LIN {X 0,Y 390.194,Z 575.883,A -85,B 0,C 180,E1 -11776.561,E2 -11776.561} C_VEL
LIN {X 0,Y 390.177,Z 575.881,A -85,B 0,C 180,E1 -11779.622,E2 -11779.622} C_VEL
LIN {X 0,Y 390.318,Z 575.868,A -85,B 0,C 180,E1 -11782.758,E2 -11782.758} C_VEL
LIN {X 0,Y 390.227,Z 575.879,A -85,B 0,C 180,E1 -11784.833,E2 -11784.833} C_VEL
LIN {X 0,Y 390.302,Z 575.869,A -85,B 0,C 180,E1 -11786.838,E2 -11786.838} C_VEL
LIN {X 0,Y 393.865,Z 588.299,A -85,B 0,C 180,E1 -11787.764,E2 -11787.764} C_VEL
LIN {X 0,Y 394.826,Z 592.713,A -85,B 0,C 180,E1 -11788.139,E2 -11788.139} C_VEL
LIN {X 0,Y 394.248,Z 604.071,A -85,B 0,C 180,E1 -11789.125,E2 -11789.125} C_VEL
LIN {X 0,Y 393.57,Z 614.626,A -85,B 0,C 180,E1 -11790.281,E2 -11790.281} C_VEL
LIN {X 0,Y 392.902,Z 623.913,A -85,B 0,C 180,E1 -11791.537,E2 -11791.537} C_VEL
LIN {X 0,Y 392.271,Z 631.723,A -85,B 0,C 180,E1 -11792.823,E2 -11792.823} C_VEL
LIN {X 0,Y 391.686,Z 639.356,A -85,B 0,C 180,E1 -11794.372,E2 -11794.372} C_VEL
LIN {X 0,Y 391.11,Z 646.386,A -85,B 0,C 180,E1 -11796.188,E2 -11796.188} C_VEL
LIN {X 0,Y 390.744,Z 651.077,A -85,B 0,C 180,E1 -11797.752,E2 -11797.752} C_VEL
LIN {X 0,Y 390.372,Z 654.695,A -85,B 0,C 180,E1 -11799.324,E2 -11799.324} C_VEL
LIN {X 0,Y 390.242,Z 656.548,A -85,B 0,C 180,E1 -11800.374,E2 -11800.374} C_VEL
LIN {X 0,Y 390.13,Z 658.928,A -85,B 0,C 180,E1 -11802.483,E2 -11802.483} C_VEL
LIN {X 0,Y 390.103,Z 659.542,A -85,B 0,C 180,E1 -11803.544,E2 -11803.544} C_VEL
LIN {X 0,Y 390.097,Z 659.724,A -85,B 0,C 180,E1 -11804.608,E2 -11804.608} C_VEL
LIN {X 0,Y 390.166,Z 659.488,A -85,B 0,C 180,E1 -11805.675,E2 -11805.675} C_VEL
LIN {X 0,Y 390.415,Z 658.214,A -85,B 0,C 180,E1 -11807.434,E2 -11807.434} C_VEL
LIN {X 0,Y 390.691,Z 656.292,A -85,B 0,C 180,E1 -11808.891,E2 -11808.891} C_VEL
LIN {X 0,Y 391.12,Z 653.303,A -85,B 0,C 180,E1 -11810.453,E2 -11810.453} C_VEL
LIN {X 0,Y 391.676,Z 648.912,A -85,B 0,C 180,E1 -11812.135,E2 -11812.135} C_VEL
LIN {X 0,Y 392.326,Z 643.825,A -85,B 0,C 180,E1 -11813.641,E2 -11813.641} C_VEL
LIN {X 0,Y 393.055,Z 637.573,A -85,B 0,C 180,E1 -11815.128,E2 -11815.128} C_VEL
LIN {X 0,Y 393.264,Z 635.478,A -85,B 0,C 180,E1 -11815.565,E2 -11815.565} C_VEL
LIN {X 0,Y 392.975,Z 632.072,A -85,B 0,C 180,E1 -11816.264,E2 -11816.264} C_VEL
LIN {X 0,Y 390.853,Z 626.407,A -85,B 0,C 180,E1 -11817.415,E2 -11817.415} C_VEL
LIN {X 0,Y 388.824,Z 620.184,A -85,B 0,C 180,E1 -11818.508,E2 -11818.508} C_VEL
LIN {X 0,Y 388.669,Z 615.858,A -85,B 0,C 180,E1 -11819.107,E2 -11819.107} C_VEL
LIN {X 0,Y 389.493,Z 606.667,A -85,B 0,C 180,E1 -11820.139,E2 -11820.139} C_VEL
LIN {X 0,Y 390.053,Z 597.639,A -85,B 0,C 180,E1 -11820.98,E2 -11820.98} C_VEL
LIN {X 0,Y 386.897,Z 587.664,A -85,B 0,C 180,E1 -11821.982,E2 -11821.982} C_VEL
LIN {X 0,Y 383.009,Z 576.778,A -85,B 0,C 180,E1 -11822.925,E2 -11822.925} C_VEL
LIN {X 0,Y 383.03,Z 576.776,A -85,B 0,C 180,E1 -11826.165,E2 -11826.165} C_VEL
LIN {X 0,Y 383.104,Z 576.928,A -85,B 0,C 180,E1 -11827.347,E2 -11827.347} C_VEL
LIN {X 0,Y 384.275,Z 584.145,A -85,B 0,C 180,E1 -11830.484,E2 -11830.484} C_VEL
LIN {X 0,Y 384.388,Z 589.077,A -85,B 0,C 180,E1 -11832.568,E2 -11832.568} C_VEL
LIN {X 0,Y 384.165,Z 597.22,A -85,B 0,C 180,E1 -11835.959,E2 -11835.959} C_VEL
LIN {X 0,Y 383.806,Z 605.658,A -85,B 0,C 180,E1 -11839.455,E2 -11839.455} C_VEL
LIN {X 0,Y 383.586,Z 613.717,A -85,B 0,C 180,E1 -11842.799,E2 -11842.799} C_VEL
LIN {X 0,Y 383.345,Z 621.722,A -85,B 0,C 180,E1 -11846.104,E2 -11846.104} C_VEL
LIN {X 0,Y 383.107,Z 627.878,A -85,B 0,C 180,E1 -11848.627,E2 -11848.627} C_VEL
LIN {X 0,Y 386.206,Z 643.214,A -85,B 0,C 180,E1 -11849.33,E2 -11849.33} C_VEL
LIN {X 0,Y 387.553,Z 651.071,A -85,B 0,C 180,E1 -11849.787,E2 -11849.787} C_VEL
LIN {X 0,Y 386.823,Z 664.164,A -85,B 0,C 180,E1 -11850.624,E2 -11850.624} C_VEL
LIN {X 0,Y 386.035,Z 675.878,A -85,B 0,C 180,E1 -11851.601,E2 -11851.601} C_VEL
LIN {X 0,Y 385.206,Z 686.528,A -85,B 0,C 180,E1 -11852.717,E2 -11852.717} C_VEL
LIN {X 0,Y 384.455,Z 696.334,A -85,B 0,C 180,E1 -11853.978,E2 -11853.978} C_VEL
LIN {X 0,Y 383.72,Z 705.192,A -85,B 0,C 180,E1 -11855.376,E2 -11855.376} C_VEL
LIN {X 0,Y 383.032,Z 713.063,A -85,B 0,C 180,E1 -11856.901,E2 -11856.901} C_VEL
LIN {X 0,Y 382.625,Z 719.518,A -85,B 0,C 180,E1 -11858.448,E2 -11858.448} C_VEL
LIN {X 0,Y 382.193,Z 725.168,A -85,B 0,C 180,E1 -11860.148,E2 -11860.148} C_VEL
LIN {X 0,Y 381.951,Z 729.276,A -85,B 0,C 180,E1 -11861.772,E2 -11861.772} C_VEL
LIN {X 0,Y 381.781,Z 731.954,A -85,B 0,C 180,E1 -11863.179,E2 -11863.179} C_VEL
LIN {X 0,Y 381.595,Z 734.309,A -85,B 0,C 180,E1 -11865.058,E2 -11865.058} C_VEL
LIN {X 0,Y 381.595,Z 735.066,A -85,B 0,C 180,E1 -11866.148,E2 -11866.148} C_VEL
LIN {X 0,Y 381.665,Z 735.426,A -85,B 0,C 180,E1 -11867.401,E2 -11867.401} C_VEL
LIN {X 0,Y 381.711,Z 734.762,A -85,B 0,C 180,E1 -11869.391,E2 -11869.391} C_VEL
LIN {X 0,Y 381.807,Z 733.822,A -85,B 0,C 180,E1 -11870.465,E2 -11870.465} C_VEL
LIN {X 0,Y 381.983,Z 732.444,A -85,B 0,C 180,E1 -11871.536,E2 -11871.536} C_VEL
LIN {X 0,Y 382.276,Z 729.651,A -85,B 0,C 180,E1 -11873.094,E2 -11873.094} C_VEL
LIN {X 0,Y 382.601,Z 725.627,A -85,B 0,C 180,E1 -11874.731,E2 -11874.731} C_VEL
LIN {X 0,Y 383.088,Z 720.539,A -85,B 0,C 180,E1 -11876.319,E2 -11876.319} C_VEL
LIN {X 0,Y 383.752,Z 714.152,A -85,B 0,C 180,E1 -11877.901,E2 -11877.901} C_VEL
LIN {X 0,Y 384.642,Z 706.243,A -85,B 0,C 180,E1 -11879.477,E2 -11879.477} C_VEL
LIN {X 0,Y 385.687,Z 696.35,A -85,B 0,C 180,E1 -11881.045,E2 -11881.045} C_VEL
LIN {X 0,Y 386.771,Z 685.973,A -85,B 0,C 180,E1 -11882.37,E2 -11882.37} C_VEL
LIN {X 0,Y 387.773,Z 675.189,A -85,B 0,C 180,E1 -11883.471,E2 -11883.471} C_VEL
LIN {X 0,Y 388.738,Z 663.277,A -85,B 0,C 180,E1 -11884.441,E2 -11884.441} C_VEL
LIN {X 0,Y 389.311,Z 652.449,A -85,B 0,C 180,E1 -11885.138,E2 -11885.138} C_VEL
LIN {X 0,Y 386.453,Z 639.446,A -85,B 0,C 180,E1 -11885.986,E2 -11885.986} C_VEL
LIN {X 0,Y 383.962,Z 630.709,A -85,B 0,C 180,E1 -11886.503,E2 -11886.503} C_VEL
LIN {X 0,Y 384.34,Z 622.273,A -85,B 0,C 180,E1 -11890.004,E2 -11890.004} C_VEL
LIN {X 0,Y 384.729,Z 613.228,A -85,B 0,C 180,E1 -11893.738,E2 -11893.738} C_VEL
LIN {X 0,Y 385.107,Z 605.416,A -85,B 0,C 180,E1 -11896.978,E2 -11896.978} C_VEL
LIN {X 0,Y 385.498,Z 597.363,A -85,B 0,C 180,E1 -11900.267,E2 -11900.267} C_VEL
LIN {X 0,Y 385.705,Z 591.791,A -85,B 0,C 180,E1 -11902.498,E2 -11902.498} C_VEL
LIN {X 0,Y 385.438,Z 587.576,A -85,B 0,C 180,E1 -11904.263,E2 -11904.263} C_VEL
LIN {X 0,Y 384.102,Z 580.962,A -85,B 0,C 180,E1 -11907.222,E2 -11907.222} C_VEL
LIN {X 0,Y 383.005,Z 576.778,A -85,B 0,C 180,E1 -11909.246,E2 -11909.246} C_VEL
LIN {X 0,Y 382.983,Z 576.781,A -85,B 0,C 180,E1 -11912.424,E2 -11912.424} C_VEL
LIN {X 0,Y 383.022,Z 576.777,A -85,B 0,C 180,E1 -11915.956,E2 -11915.956} C_VEL
LIN {X 0,Y 383.018,Z 576.776,A -85,B 0,C 180,E1 -11919.589,E2 -11919.589} C_VEL
LIN {X 0,Y 383.061,Z 576.765,A -85,B 0,C 180,E1 -11922.79,E2 -11922.79} C_VEL
LIN {X 0,Y 383.074,Z 576.773,A -85,B 0,C 180,E1 -11924.108,E2 -11924.108} C_VEL
LIN {X 0,Y 384.746,Z 584.934,A -85,B 0,C 180,E1 -11927.48,E2 -11927.48} C_VEL
LIN {X 0,Y 386.352,Z 592.664,A -85,B 0,C 180,E1 -11930.457,E2 -11930.457} C_VEL
LIN {X 0,Y 387.193,Z 598.391,A -85,B 0,C 180,E1 -11932.514,E2 -11932.514} C_VEL
LIN {X 0,Y 386.751,Z 604.218,A -85,B 0,C 180,E1 -11934.445,E2 -11934.445} C_VEL
LIN {X 0,Y 385.518,Z 615.731,A -85,B 0,C 180,E1 -11938.086,E2 -11938.086} C_VEL
LIN {X 0,Y 384.539,Z 627.309,A -85,B 0,C 180,E1 -11941.63,E2 -11941.63} C_VEL
LIN {X 0,Y 383.716,Z 638.912,A -85,B 0,C 180,E1 -11945.087,E2 -11945.087} C_VEL
LIN {X 0,Y 383.048,Z 650.507,A -85,B 0,C 180,E1 -11948.474,E2 -11948.474} C_VEL
LIN {X 0,Y 382.761,Z 657.07,A -85,B 0,C 180,E1 -11950.353,E2 -11950.353} C_VEL
LIN {X 0,Y 385.272,Z 672.356,A -85,B 0,C 180,E1 -11951.017,E2 -11951.017} C_VEL
LIN {X 0,Y 386.439,Z 685.505,A -85,B 0,C 180,E1 -11951.617,E2 -11951.617} C_VEL
LIN {X 0,Y 386.921,Z 699.026,A -85,B 0,C 180,E1 -11952.425,E2 -11952.425} C_VEL
LIN {X 0,Y 387.037,Z 706.618,A -85,B 0,C 180,E1 -11952.975,E2 -11952.975} C_VEL
LIN {X 0,Y 385.965,Z 718.985,A -85,B 0,C 180,E1 -11954.015,E2 -11954.015} C_VEL
LIN {X 0,Y 384.927,Z 730.191,A -85,B 0,C 180,E1 -11955.191,E2 -11955.191} C_VEL
LIN {X 0,Y 383.955,Z 740.244,A -85,B 0,C 180,E1 -11956.505,E2 -11956.505} C_VEL
LIN {X 0,Y 383.178,Z 750.058,A -85,B 0,C 180,E1 -11958.093,E2 -11958.093} C_VEL
LIN {X 0,Y 382.524,Z 757.933,A -85,B 0,C 180,E1 -11959.682,E2 -11959.682} C_VEL
LIN {X 0,Y 382.11,Z 765.236,A -85,B 0,C 180,E1 -11961.54,E2 -11961.54} C_VEL
LIN {X 0,Y 381.865,Z 770.115,A -85,B 0,C 180,E1 -11963.13,E2 -11963.13} C_VEL
LIN {X 0,Y 381.825,Z 773.852,A -85,B 0,C 180,E1 -11964.721,E2 -11964.721} C_VEL
LIN {X 0,Y 381.768,Z 775.736,A -85,B 0,C 180,E1 -11965.778,E2 -11965.778} C_VEL
LIN {X 0,Y 381.769,Z 777.178,A -85,B 0,C 180,E1 -11966.835,E2 -11966.835} C_VEL
LIN {X 0,Y 381.862,Z 778.213,A -85,B 0,C 180,E1 -11967.892,E2 -11967.892} C_VEL
LIN {X 0,Y 381.847,Z 778.806,A -85,B 0,C 180,E1 -11968.946,E2 -11968.946} C_VEL
LIN {X 0,Y 381.869,Z 778.946,A -85,B 0,C 180,E1 -11970.001,E2 -11970.001} C_VEL
LIN {X 0,Y 381.858,Z 778.675,A -85,B 0,C 180,E1 -11971.056,E2 -11971.056} C_VEL
LIN {X 0,Y 381.865,Z 777.996,A -85,B 0,C 180,E1 -11972.11,E2 -11972.11} C_VEL
LIN {X 0,Y 381.787,Z 776.839,A -85,B 0,C 180,E1 -11973.167,E2 -11973.167} C_VEL
LIN {X 0,Y 381.83,Z 774.298,A -85,B 0,C 180,E1 -11974.752,E2 -11974.752} C_VEL
LIN {X 0,Y 381.82,Z 770.678,A -85,B 0,C 180,E1 -11976.342,E2 -11976.342} C_VEL
LIN {X 0,Y 381.995,Z 765.892,A -85,B 0,C 180,E1 -11977.932,E2 -11977.932} C_VEL
LIN {X 0,Y 382.281,Z 759.797,A -85,B 0,C 180,E1 -11979.525,E2 -11979.525} C_VEL
LIN {X 0,Y 382.71,Z 752.184,A -85,B 0,C 180,E1 -11981.118,E2 -11981.118} C_VEL
LIN {X 0,Y 383.322,Z 744.375,A -85,B 0,C 180,E1 -11982.442,E2 -11982.442} C_VEL
LIN {X 0,Y 384.079,Z 734.843,A -85,B 0,C 180,E1 -11983.762,E2 -11983.762} C_VEL
LIN {X 0,Y 384.805,Z 724.318,A -85,B 0,C 180,E1 -11984.951,E2 -11984.951} C_VEL
LIN {X 0,Y 385.646,Z 712.566,A -85,B 0,C 180,E1 -11986.001,E2 -11986.001} C_VEL
LIN {X 0,Y 386.215,Z 702.349,A -85,B 0,C 180,E1 -11986.724,E2 -11986.724} C_VEL
LIN {X 0,Y 385.424,Z 690.737,A -85,B 0,C 180,E1 -11987.404,E2 -11987.404} C_VEL
LIN {X 0,Y 384.39,Z 677.083,A -85,B 0,C 180,E1 -11987.988,E2 -11987.988} C_VEL
LIN {X 0,Y 382.604,Z 659.203,A -85,B 0,C 180,E1 -11988.578,E2 -11988.578} C_VEL
LIN {X 0,Y 383.037,Z 646.75,A -85,B 0,C 180,E1 -11992.095,E2 -11992.095} C_VEL
LIN {X 0,Y 383.619,Z 634.832,A -85,B 0,C 180,E1 -11995.502,E2 -11995.502} C_VEL
LIN {X 0,Y 384.342,Z 624.02,A -85,B 0,C 180,E1 -11998.631,E2 -11998.631} C_VEL
LIN {X 0,Y 385.107,Z 612.782,A -85,B 0,C 180,E1 -12001.955,E2 -12001.955} C_VEL
LIN {X 0,Y 386.026,Z 601.856,A -85,B 0,C 180,E1 -12005.247,E2 -12005.247} C_VEL
LIN {X 0,Y 386.431,Z 595.525,A -85,B 0,C 180,E1 -12007.209,E2 -12007.209} C_VEL
LIN {X 0,Y 385.417,Z 589.088,A -85,B 0,C 180,E1 -12009.343,E2 -12009.343} C_VEL
LIN {X 0,Y 383.551,Z 579.507,A -85,B 0,C 180,E1 -12012.686,E2 -12012.686} C_VEL
LIN {X 0,Y 383.025,Z 576.776,A -85,B 0,C 180,E1 -12013.735,E2 -12013.735} C_VEL
LIN {X 0,Y 383.015,Z 576.777,A -85,B 0,C 180,E1 -12017.24,E2 -12017.24} C_VEL
LIN {X 0,Y 383.021,Z 576.776,A -85,B 0,C 180,E1 -12020.413,E2 -12020.413} C_VEL
LIN {X 0,Y 383.032,Z 576.774,A -85,B 0,C 180,E1 -12024.045,E2 -12024.045} C_VEL
LIN {X 0,Y 382.992,Z 576.776,A -85,B 0,C 180,E1 -12027.578,E2 -12027.578} C_VEL
LIN {X 0,Y 382.997,Z 576.78,A -85,B 0,C 180,E1 -12030.3,E2 -12030.3} C_VEL
LIN {X 0,Y 383.085,Z 576.768,A -85,B 0,C 180,E1 -12034.021,E2 -12034.021} C_VEL
LIN {X 0,Y 383.013,Z 576.773,A -85,B 0,C 180,E1 -12037.335,E2 -12037.335} C_VEL
LIN {X 0,Y 383.065,Z 576.769,A -85,B 0,C 180,E1 -12040.716,E2 -12040.716} C_VEL
LIN {X 0,Y 383.085,Z 576.767,A -85,B 0,C 180,E1 -12044.026,E2 -12044.026} C_VEL
LIN {X 0,Y 383.141,Z 576.757,A -85,B 0,C 180,E1 -12047.284,E2 -12047.284} C_VEL
LIN {X 0,Y 383.156,Z 576.76,A -85,B 0,C 180,E1 -12050.498,E2 -12050.498} C_VEL
LIN {X 0,Y 383.278,Z 576.744,A -85,B 0,C 180,E1 -12052.625,E2 -12052.625} C_VEL
LIN {X 0,Y 383.202,Z 576.752,A -85,B 0,C 180,E1 -12054.738,E2 -12054.738} C_VEL
LIN {X 0,Y 383.389,Z 576.728,A -85,B 0,C 180,E1 -12057.899,E2 -12057.899} C_VEL
LIN {X 0,Y 383.524,Z 576.712,A -85,B 0,C 180,E1 -12060,E2 -12060} C_VEL
LIN {X 0,Y 383.249,Z 576.744,A -85,B 0,C 180,E1 -12063.153,E2 -12063.153} C_VEL
LIN {X 0,Y 383.273,Z 576.742,A -85,B 0,C 180,E1 -12066.632,E2 -12066.632} C_VEL
LIN {X 0,Y 383.264,Z 576.747,A -85,B 0,C 180,E1 -12068.435,E2 -12068.435} C_VEL
LIN {X 0,Y 383.1,Z 576.762,A -85,B 0,C 180,E1 -12071.642,E2 -12071.642} C_VEL
LIN {X 0,Y 383.113,Z 576.763,A -85,B 0,C 180,E1 -12074.881,E2 -12074.881} C_VEL
LIN {X 0,Y 383.092,Z 576.767,A -85,B 0,C 180,E1 -12078.172,E2 -12078.172} C_VEL
LIN {X 0,Y 382.996,Z 576.775,A -85,B 0,C 180,E1 -12081.53,E2 -12081.53} C_VEL
LIN {X 0,Y 383.055,Z 576.769,A -85,B 0,C 180,E1 -12084.96,E2 -12084.96} C_VEL
LIN {X 0,Y 383.043,Z 576.774,A -85,B 0,C 180,E1 -12088.492,E2 -12088.492} C_VEL
LIN {X 0,Y 383.011,Z 576.777,A -85,B 0,C 180,E1 -12092.149,E2 -12092.149} C_VEL
LIN {X 0,Y 383.02,Z 576.776,A -85,B 0,C 180,E1 -12094.667,E2 -12094.667} C_VEL
LIN {X 0,Y 383.003,Z 576.776,A -85,B 0,C 180,E1 -12097.903,E2 -12097.903} C_VEL
LIN {X 0,Y 382.986,Z 576.776,A -85,B 0,C 180,E1 -12101.347,E2 -12101.347} C_VEL
LIN {X 0,Y 383.001,Z 576.779,A -85,B 0,C 180,E1 -12104.303,E2 -12104.303} C_VEL
LIN {X 0,Y 383.011,Z 576.773,A -85,B 0,C 180,E1 -12107.239,E2 -12107.239} C_VEL
LIN {X 0,Y 383.017,Z 576.778,A -85,B 0,C 180,E1 -12110.413,E2 -12110.413} C_VEL
LIN {X 0,Y 383.025,Z 576.773,A -85,B 0,C 180,E1 -12114.044,E2 -12114.044} C_VEL
LIN {X 0,Y 382.987,Z 576.776,A -85,B 0,C 180,E1 -12117.577,E2 -12117.577} C_VEL
LIN {X 0,Y 382.993,Z 576.78,A -85,B 0,C 180,E1 -12120.299,E2 -12120.299} C_VEL
LIN {X 0,Y 383.08,Z 576.766,A -85,B 0,C 180,E1 -12124.02,E2 -12124.02} C_VEL
LIN {X 0,Y 383.013,Z 576.773,A -85,B 0,C 180,E1 -12127.335,E2 -12127.335} C_VEL
LIN {X 0,Y 383.06,Z 576.772,A -85,B 0,C 180,E1 -12130.715,E2 -12130.715} C_VEL
LIN {X 0,Y 383.081,Z 576.766,A -85,B 0,C 180,E1 -12134.026,E2 -12134.026} C_VEL
LIN {X 0,Y 383.141,Z 576.757,A -85,B 0,C 180,E1 -12137.283,E2 -12137.283} C_VEL
LIN {X 0,Y 383.156,Z 576.76,A -85,B 0,C 180,E1 -12140.497,E2 -12140.497} C_VEL
LIN {X 0,Y 383.273,Z 576.746,A -85,B 0,C 180,E1 -12142.624,E2 -12142.624} C_VEL
LIN {X 0,Y 383.199,Z 576.755,A -85,B 0,C 180,E1 -12144.738,E2 -12144.738} C_VEL
LIN {X 0,Y 383.222,Z 576.898,A -85,B 0,C 180,E1 -12146.582,E2 -12146.582} C_VEL
LIN {X 0,Y 386.654,Z 588.417,A -85,B 0,C 180,E1 -12147.447,E2 -12147.447} C_VEL
LIN {X 0,Y 387.963,Z 593.955,A -85,B 0,C 180,E1 -12147.923,E2 -12147.923} C_VEL
LIN {X 0,Y 387.324,Z 605.582,A -85,B 0,C 180,E1 -12148.959,E2 -12148.959} C_VEL
LIN {X 0,Y 386.584,Z 616.832,A -85,B 0,C 180,E1 -12150.234,E2 -12150.234} C_VEL
LIN {X 0,Y 385.88,Z 626.232,A -85,B 0,C 180,E1 -12151.565,E2 -12151.565} C_VEL
LIN {X 0,Y 385.118,Z 635.143,A -85,B 0,C 180,E1 -12153.137,E2 -12153.137} C_VEL
LIN {X 0,Y 384.551,Z 642.319,A -85,B 0,C 180,E1 -12154.716,E2 -12154.716} C_VEL
LIN {X 0,Y 384.059,Z 648.085,A -85,B 0,C 180,E1 -12156.303,E2 -12156.303} C_VEL
LIN {X 0,Y 383.645,Z 653.091,A -85,B 0,C 180,E1 -12158.092,E2 -12158.092} C_VEL
LIN {X 0,Y 383.326,Z 656.112,A -85,B 0,C 180,E1 -12159.497,E2 -12159.497} C_VEL
LIN {X 0,Y 383.182,Z 657.847,A -85,B 0,C 180,E1 -12160.567,E2 -12160.567} C_VEL
LIN {X 0,Y 383.102,Z 660.105,A -85,B 0,C 180,E1 -12162.716,E2 -12162.716} C_VEL
LIN {X 0,Y 383.09,Z 660.617,A -85,B 0,C 180,E1 -12163.796,E2 -12163.796} C_VEL
LIN {X 0,Y 383.179,Z 660.422,A -85,B 0,C 180,E1 -12165.968,E2 -12165.968} C_VEL
LIN {X 0,Y 383.425,Z 659.173,A -85,B 0,C 180,E1 -12167.612,E2 -12167.612} C_VEL
LIN {X 0,Y 383.909,Z 656.009,A -85,B 0,C 180,E1 -12169.795,E2 -12169.795} C_VEL
LIN {X 0,Y 384.472,Z 652.376,A -85,B 0,C 180,E1 -12171.443,E2 -12171.443} C_VEL
LIN {X 0,Y 385.091,Z 647.543,A -85,B 0,C 180,E1 -12173.101,E2 -12173.101} C_VEL
LIN {X 0,Y 385.893,Z 641.333,A -85,B 0,C 180,E1 -12174.763,E2 -12174.763} C_VEL
LIN {X 0,Y 386.677,Z 634.882,A -85,B 0,C 180,E1 -12176.151,E2 -12176.151} C_VEL
LIN {X 0,Y 387.637,Z 626.735,A -85,B 0,C 180,E1 -12177.583,E2 -12177.583} C_VEL
LIN {X 0,Y 388.549,Z 617.215,A -85,B 0,C 180,E1 -12178.936,E2 -12178.936} C_VEL
LIN {X 0,Y 388.669,Z 615.858,A -85,B 0,C 180,E1 -12179.107,E2 -12179.107} C_VEL
LIN {X 0,Y 388.549,Z 611.371,A -85,B 0,C 180,E1 -12179.682,E2 -12179.682} C_VEL
LIN {X 0,Y 387.464,Z 606.988,A -85,B 0,C 180,E1 -12180.26,E2 -12180.26} C_VEL
LIN {X 0,Y 383.752,Z 598.255,A -85,B 0,C 180,E1 -12181.375,E2 -12181.375} C_VEL
LIN {X 0,Y 381.165,Z 592.074,A -85,B 0,C 180,E1 -12182.058,E2 -12182.058} C_VEL
LIN {X 0,Y 376.937,Z 580.449,A -85,B 0,C 180,E1 -12183.142,E2 -12183.142} C_VEL
LIN {X 0,Y 375.967,Z 577.651,A -85,B 0,C 180,E1 -12183.388,E2 -12183.388} C_VEL
LIN {X 0,Y 376.018,Z 577.726,A -85,B 0,C 180,E1 -12187.067,E2 -12187.067} C_VEL
LIN {X 0,Y 376.947,Z 582.925,A -85,B 0,C 180,E1 -12189.338,E2 -12189.338} C_VEL
LIN {X 0,Y 377.423,Z 587.324,A -85,B 0,C 180,E1 -12191.262,E2 -12191.262} C_VEL
LIN {X 0,Y 377.283,Z 594.399,A -85,B 0,C 180,E1 -12194.245,E2 -12194.245} C_VEL
LIN {X 0,Y 377.045,Z 601.499,A -85,B 0,C 180,E1 -12197.232,E2 -12197.232} C_VEL
LIN {X 0,Y 376.686,Z 610.934,A -85,B 0,C 180,E1 -12201.165,E2 -12201.165} C_VEL
LIN {X 0,Y 376.45,Z 617.747,A -85,B 0,C 180,E1 -12204.011,E2 -12204.011} C_VEL
LIN {X 0,Y 376.186,Z 625.456,A -85,B 0,C 180,E1 -12207.212,E2 -12207.212} C_VEL
LIN {X 0,Y 376.062,Z 628.224,A -85,B 0,C 180,E1 -12208.349,E2 -12208.349} C_VEL
LIN {X 0,Y 378.816,Z 641.666,A -85,B 0,C 180,E1 -12208.958,E2 -12208.958} C_VEL
LIN {X 0,Y 380.616,Z 652.004,A -85,B 0,C 180,E1 -12209.566,E2 -12209.566} C_VEL
LIN {X 0,Y 379.931,Z 664.52,A -85,B 0,C 180,E1 -12210.387,E2 -12210.387} C_VEL
LIN {X 0,Y 379.142,Z 675.802,A -85,B 0,C 180,E1 -12211.339,E2 -12211.339} C_VEL
LIN {X 0,Y 378.207,Z 687.494,A -85,B 0,C 180,E1 -12212.589,E2 -12212.589} C_VEL
LIN {X 0,Y 377.508,Z 696.398,A -85,B 0,C 180,E1 -12213.759,E2 -12213.759} C_VEL
LIN {X 0,Y 376.75,Z 705.338,A -85,B 0,C 180,E1 -12215.184,E2 -12215.184} C_VEL
LIN {X 0,Y 375.979,Z 713.947,A -85,B 0,C 180,E1 -12216.888,E2 -12216.888} C_VEL
LIN {X 0,Y 375.486,Z 720.801,A -85,B 0,C 180,E1 -12218.594,E2 -12218.594} C_VEL
LIN {X 0,Y 375.099,Z 726.125,A -85,B 0,C 180,E1 -12220.291,E2 -12220.291} C_VEL
LIN {X 0,Y 374.857,Z 730.176,A -85,B 0,C 180,E1 -12221.98,E2 -12221.98} C_VEL
LIN {X 0,Y 374.626,Z 733.075,A -85,B 0,C 180,E1 -12223.657,E2 -12223.657} C_VEL
LIN {X 0,Y 374.517,Z 734.435,A -85,B 0,C 180,E1 -12224.769,E2 -12224.769} C_VEL
LIN {X 0,Y 374.523,Z 735.326,A -85,B 0,C 180,E1 -12225.881,E2 -12225.881} C_VEL
LIN {X 0,Y 374.573,Z 735.843,A -85,B 0,C 180,E1 -12227.326,E2 -12227.326} C_VEL
LIN {X 0,Y 374.634,Z 735.409,A -85,B 0,C 180,E1 -12229.188,E2 -12229.188} C_VEL
LIN {X 0,Y 374.726,Z 734.566,A -85,B 0,C 180,E1 -12230.283,E2 -12230.283} C_VEL
LIN {X 0,Y 374.877,Z 733.322,A -85,B 0,C 180,E1 -12231.375,E2 -12231.375} C_VEL
LIN {X 0,Y 375.208,Z 730.488,A -85,B 0,C 180,E1 -12233.079,E2 -12233.079} C_VEL
LIN {X 0,Y 375.537,Z 726.908,A -85,B 0,C 180,E1 -12234.631,E2 -12234.631} C_VEL
LIN {X 0,Y 376.031,Z 722.067,A -85,B 0,C 180,E1 -12236.25,E2 -12236.25} C_VEL
LIN {X 0,Y 376.71,Z 715.951,A -85,B 0,C 180,E1 -12237.862,E2 -12237.862} C_VEL
LIN {X 0,Y 377.614,Z 708.356,A -85,B 0,C 180,E1 -12239.467,E2 -12239.467} C_VEL
LIN {X 0,Y 378.71,Z 698.979,A -85,B 0,C 180,E1 -12241.064,E2 -12241.064} C_VEL
LIN {X 0,Y 379.853,Z 688.639,A -85,B 0,C 180,E1 -12242.462,E2 -12242.462} C_VEL
LIN {X 0,Y 380.937,Z 678.1,A -85,B 0,C 180,E1 -12243.615,E2 -12243.615} C_VEL
LIN {X 0,Y 381.939,Z 666.592,A -85,B 0,C 180,E1 -12244.617,E2 -12244.617} C_VEL
LIN {X 0,Y 382.814,Z 655.046,A -85,B 0,C 180,E1 -12245.408,E2 -12245.408} C_VEL
LIN {X 0,Y 380.548,Z 643.229,A -85,B 0,C 180,E1 -12246.243,E2 -12246.243} C_VEL
LIN {X 0,Y 377.646,Z 633.194,A -85,B 0,C 180,E1 -12246.875,E2 -12246.875} C_VEL
LIN {X 0,Y 377.088,Z 631.131,A -85,B 0,C 180,E1 -12247.026,E2 -12247.026} C_VEL
LIN {X 0,Y 377.464,Z 623.623,A -85,B 0,C 180,E1 -12250.189,E2 -12250.189} C_VEL
LIN {X 0,Y 377.88,Z 614.56,A -85,B 0,C 180,E1 -12253.992,E2 -12253.992} C_VEL
LIN {X 0,Y 378.322,Z 606.751,A -85,B 0,C 180,E1 -12257.292,E2 -12257.292} C_VEL
LIN {X 0,Y 378.873,Z 597.387,A -85,B 0,C 180,E1 -12261.206,E2 -12261.206} C_VEL
LIN {X 0,Y 378.933,Z 591.827,A -85,B 0,C 180,E1 -12263.501,E2 -12263.501} C_VEL
LIN {X 0,Y 378.15,Z 586.514,A -85,B 0,C 180,E1 -12265.897,E2 -12265.897} C_VEL
LIN {X 0,Y 376.595,Z 580.008,A -85,B 0,C 180,E1 -12269.027,E2 -12269.027} C_VEL
LIN {X 0,Y 375.963,Z 577.655,A -85,B 0,C 180,E1 -12270.313,E2 -12270.313} C_VEL
LIN {X 0,Y 375.954,Z 577.656,A -85,B 0,C 180,E1 -12274.112,E2 -12274.112} C_VEL
LIN {X 0,Y 375.95,Z 577.655,A -85,B 0,C 180,E1 -12276.742,E2 -12276.742} C_VEL
LIN {X 0,Y 375.995,Z 577.649,A -85,B 0,C 180,E1 -12279.974,E2 -12279.974} C_VEL
LIN {X 0,Y 376.036,Z 577.656,A -85,B 0,C 180,E1 -12283.591,E2 -12283.591} C_VEL
LIN {X 0,Y 377.496,Z 584.616,A -85,B 0,C 180,E1 -12286.559,E2 -12286.559} C_VEL
LIN {X 0,Y 379.411,Z 593.974,A -85,B 0,C 180,E1 -12290.28,E2 -12290.28} C_VEL
LIN {X 0,Y 380.274,Z 599.775,A -85,B 0,C 180,E1 -12292.42,E2 -12292.42} C_VEL
LIN {X 0,Y 379.726,Z 606.051,A -85,B 0,C 180,E1 -12294.524,E2 -12294.524} C_VEL
LIN {X 0,Y 378.525,Z 616.968,A -85,B 0,C 180,E1 -12298.053,E2 -12298.053} C_VEL
LIN {X 0,Y 377.504,Z 628.495,A -85,B 0,C 180,E1 -12301.659,E2 -12301.659} C_VEL
LIN {X 0,Y 376.638,Z 640.044,A -85,B 0,C 180,E1 -12305.176,E2 -12305.176} C_VEL
LIN {X 0,Y 375.929,Z 651.604,A -85,B 0,C 180,E1 -12308.621,E2 -12308.621} C_VEL
LIN {X 0,Y 375.812,Z 655.399,A -85,B 0,C 180,E1 -12309.727,E2 -12309.727} C_VEL
LIN {X 0,Y 376.154,Z 658.371,A -85,B 0,C 180,E1 -12309.952,E2 -12309.952} C_VEL
LIN {X 0,Y 378.769,Z 673.448,A -85,B 0,C 180,E1 -12310.617,E2 -12310.617} C_VEL
LIN {X 0,Y 379.78,Z 685.985,A -85,B 0,C 180,E1 -12311.235,E2 -12311.235} C_VEL
LIN {X 0,Y 380.207,Z 699.87,A -85,B 0,C 180,E1 -12312.104,E2 -12312.104} C_VEL
LIN {X 0,Y 380.303,Z 707.215,A -85,B 0,C 180,E1 -12312.664,E2 -12312.664} C_VEL
LIN {X 0,Y 379.167,Z 719.364,A -85,B 0,C 180,E1 -12313.72,E2 -12313.72} C_VEL
LIN {X 0,Y 378.06,Z 730.335,A -85,B 0,C 180,E1 -12314.916,E2 -12314.916} C_VEL
LIN {X 0,Y 377.034,Z 740.221,A -85,B 0,C 180,E1 -12316.252,E2 -12316.252} C_VEL
LIN {X 0,Y 376.215,Z 749.941,A -85,B 0,C 180,E1 -12317.869,E2 -12317.869} C_VEL
LIN {X 0,Y 375.475,Z 757.745,A -85,B 0,C 180,E1 -12319.486,E2 -12319.486} C_VEL
LIN {X 0,Y 375.048,Z 765.014,A -85,B 0,C 180,E1 -12321.379,E2 -12321.379} C_VEL
LIN {X 0,Y 374.802,Z 769.841,A -85,B 0,C 180,E1 -12323,E2 -12323} C_VEL
LIN {X 0,Y 374.72,Z 773.528,A -85,B 0,C 180,E1 -12324.62,E2 -12324.62} C_VEL
LIN {X 0,Y 374.691,Z 775.383,A -85,B 0,C 180,E1 -12325.698,E2 -12325.698} C_VEL
LIN {X 0,Y 374.791,Z 777.833,A -85,B 0,C 180,E1 -12327.852,E2 -12327.852} C_VEL
LIN {X 0,Y 374.772,Z 778.394,A -85,B 0,C 180,E1 -12328.926,E2 -12328.926} C_VEL
LIN {X 0,Y 374.791,Z 778.52,A -85,B 0,C 180,E1 -12330.001,E2 -12330.001} C_VEL
LIN {X 0,Y 374.782,Z 778.234,A -85,B 0,C 180,E1 -12331.075,E2 -12331.075} C_VEL
LIN {X 0,Y 374.794,Z 777.53,A -85,B 0,C 180,E1 -12332.15,E2 -12332.15} C_VEL
LIN {X 0,Y 374.693,Z 776.342,A -85,B 0,C 180,E1 -12333.227,E2 -12333.227} C_VEL
LIN {X 0,Y 374.761,Z 773.762,A -85,B 0,C 180,E1 -12334.842,E2 -12334.842} C_VEL
LIN {X 0,Y 374.75,Z 770.096,A -85,B 0,C 180,E1 -12336.462,E2 -12336.462} C_VEL
LIN {X 0,Y 374.917,Z 765.26,A -85,B 0,C 180,E1 -12338.083,E2 -12338.083} C_VEL
LIN {X 0,Y 375.231,Z 759.11,A -85,B 0,C 180,E1 -12339.706,E2 -12339.706} C_VEL
LIN {X 0,Y 375.704,Z 751.421,A -85,B 0,C 180,E1 -12341.328,E2 -12341.328} C_VEL
LIN {X 0,Y 376.291,Z 743.515,A -85,B 0,C 180,E1 -12342.678,E2 -12342.678} C_VEL
LIN {X 0,Y 377.067,Z 733.897,A -85,B 0,C 180,E1 -12344.023,E2 -12344.023} C_VEL
LIN {X 0,Y 377.841,Z 723.273,A -85,B 0,C 180,E1 -12345.233,E2 -12345.233} C_VEL
LIN {X 0,Y 378.752,Z 711.317,A -85,B 0,C 180,E1 -12346.3,E2 -12346.3} C_VEL
LIN {X 0,Y 379.252,Z 703.044,A -85,B 0,C 180,E1 -12346.901,E2 -12346.901} C_VEL
LIN {X 0,Y 378.535,Z 691.77,A -85,B 0,C 180,E1 -12347.593,E2 -12347.593} C_VEL
LIN {X 0,Y 377.489,Z 677.548,A -85,B 0,C 180,E1 -12348.236,E2 -12348.236} C_VEL
LIN {X 0,Y 375.553,Z 658.297,A -85,B 0,C 180,E1 -12348.869,E2 -12348.869} C_VEL
LIN {X 0,Y 375.92,Z 647.564,A -85,B 0,C 180,E1 -12351.958,E2 -12351.958} C_VEL
LIN {X 0,Y 376.514,Z 635.67,A -85,B 0,C 180,E1 -12355.425,E2 -12355.425} C_VEL
LIN {X 0,Y 377.195,Z 625.849,A -85,B 0,C 180,E1 -12358.337,E2 -12358.337} C_VEL
LIN {X 0,Y 378.026,Z 614.7,A -85,B 0,C 180,E1 -12361.683,E2 -12361.683} C_VEL
LIN {X 0,Y 379.025,Z 602.849,A -85,B 0,C 180,E1 -12365.327,E2 -12365.327} C_VEL
LIN {X 0,Y 379.46,Z 596.873,A -85,B 0,C 180,E1 -12367.211,E2 -12367.211} C_VEL
LIN {X 0,Y 378.598,Z 591.165,A -85,B 0,C 180,E1 -12369.136,E2 -12369.136} C_VEL
LIN {X 0,Y 376.992,Z 582.597,A -85,B 0,C 180,E1 -12372.155,E2 -12372.155} C_VEL
LIN {X 0,Y 375.997,Z 577.652,A -85,B 0,C 180,E1 -12374.043,E2 -12374.043} C_VEL
LIN {X 0,Y 375.936,Z 577.658,A -85,B 0,C 180,E1 -12377.7,E2 -12377.7} C_VEL
LIN {X 0,Y 375.969,Z 577.654,A -85,B 0,C 180,E1 -12380.538,E2 -12380.538} C_VEL
LIN {X 0,Y 375.97,Z 577.65,A -85,B 0,C 180,E1 -12383.495,E2 -12383.495} C_VEL
LIN {X 0,Y 375.965,Z 577.653,A -85,B 0,C 180,E1 -12385.889,E2 -12385.889} C_VEL
LIN {X 0,Y 375.969,Z 577.651,A -85,B 0,C 180,E1 -12389.687,E2 -12389.687} C_VEL
LIN {X 0,Y 376.025,Z 577.643,A -85,B 0,C 180,E1 -12393.348,E2 -12393.348} C_VEL
LIN {X 0,Y 376.001,Z 577.647,A -85,B 0,C 180,E1 -12396.888,E2 -12396.888} C_VEL
LIN {X 0,Y 376.003,Z 577.651,A -85,B 0,C 180,E1 -12400.339,E2 -12400.339} C_VEL
LIN {X 0,Y 376.033,Z 577.643,A -85,B 0,C 180,E1 -12403.719,E2 -12403.719} C_VEL
LIN {X 0,Y 376.108,Z 577.634,A -85,B 0,C 180,E1 -12407.042,E2 -12407.042} C_VEL
LIN {X 0,Y 376.124,Z 577.636,A -85,B 0,C 180,E1 -12410.318,E2 -12410.318} C_VEL
LIN {X 0,Y 376.235,Z 577.622,A -85,B 0,C 180,E1 -12412.486,E2 -12412.486} C_VEL
LIN {X 0,Y 376.175,Z 577.628,A -85,B 0,C 180,E1 -12414.64,E2 -12414.64} C_VEL
LIN {X 0,Y 376.355,Z 577.604,A -85,B 0,C 180,E1 -12417.859,E2 -12417.859} C_VEL
LIN {X 0,Y 376.493,Z 577.587,A -85,B 0,C 180,E1 -12420,E2 -12420} C_VEL
LIN {X 0,Y 376.187,Z 577.623,A -85,B 0,C 180,E1 -12423.212,E2 -12423.212} C_VEL
LIN {X 0,Y 376.238,Z 577.62,A -85,B 0,C 180,E1 -12426.623,E2 -12426.623} C_VEL
LIN {X 0,Y 376.209,Z 577.625,A -85,B 0,C 180,E1 -12428.595,E2 -12428.595} C_VEL
LIN {X 0,Y 376.053,Z 577.641,A -85,B 0,C 180,E1 -12431.863,E2 -12431.863} C_VEL
LIN {X 0,Y 376.062,Z 577.639,A -85,B 0,C 180,E1 -12435.167,E2 -12435.167} C_VEL
LIN {X 0,Y 376.027,Z 577.648,A -85,B 0,C 180,E1 -12438.525,E2 -12438.525} C_VEL
LIN {X 0,Y 375.966,Z 577.652,A -85,B 0,C 180,E1 -12441.954,E2 -12441.954} C_VEL
LIN {X 0,Y 376.009,Z 577.645,A -85,B 0,C 180,E1 -12445.46,E2 -12445.46} C_VEL
LIN {X 0,Y 375.972,Z 577.651,A -85,B 0,C 180,E1 -12449.078,E2 -12449.078} C_VEL
LIN {X 0,Y 375.951,Z 577.655,A -85,B 0,C 180,E1 -12452.828,E2 -12452.828} C_VEL
LIN {X 0,Y 375.96,Z 577.651,A -85,B 0,C 180,E1 -12455.415,E2 -12455.415} C_VEL
LIN {X 0,Y 375.977,Z 577.653,A -85,B 0,C 180,E1 -12458.27,E2 -12458.27} C_VEL
LIN {X 0,Y 375.936,Z 577.654,A -85,B 0,C 180,E1 -12461.6,E2 -12461.6} C_VEL
LIN {X 0,Y 375.931,Z 577.655,A -85,B 0,C 180,E1 -12465.267,E2 -12465.267} C_VEL
LIN {X 0,Y 375.937,Z 577.659,A -85,B 0,C 180,E1 -12468.398,E2 -12468.398} C_VEL
LIN {X 0,Y 375.975,Z 577.65,A -85,B 0,C 180,E1 -12471.729,E2 -12471.729} C_VEL
LIN {X 0,Y 375.98,Z 577.649,A -85,B 0,C 180,E1 -12475.332,E2 -12475.332} C_VEL
LIN {X 0,Y 375.958,Z 577.657,A -85,B 0,C 180,E1 -12478.437,E2 -12478.437} C_VEL
LIN {X 0,Y 375.983,Z 577.651,A -85,B 0,C 180,E1 -12482.139,E2 -12482.139} C_VEL
LIN {X 0,Y 376.007,Z 577.651,A -85,B 0,C 180,E1 -12484.538,E2 -12484.538} C_VEL
LIN {X 0,Y 375.968,Z 577.652,A -85,B 0,C 180,E1 -12488.045,E2 -12488.045} C_VEL
LIN {X 0,Y 376.009,Z 577.645,A -85,B 0,C 180,E1 -12491.472,E2 -12491.472} C_VEL
LIN {X 0,Y 376.059,Z 577.643,A -85,B 0,C 180,E1 -12494.832,E2 -12494.832} C_VEL
LIN {X 0,Y 376.058,Z 577.641,A -85,B 0,C 180,E1 -12498.136,E2 -12498.136} C_VEL
LIN {X 0,Y 376.257,Z 577.615,A -85,B 0,C 180,E1 -12501.876,E2 -12501.876} C_VEL
LIN {X 0,Y 376.172,Z 577.63,A -85,B 0,C 180,E1 -12504.639,E2 -12504.639} C_VEL
LIN {X 0,Y 376.121,Z 577.635,A -85,B 0,C 180,E1 -12506.283,E2 -12506.283} C_VEL
LIN {X 0,Y 379.939,Z 590.351,A -85,B 0,C 180,E1 -12507.272,E2 -12507.272} C_VEL
LIN {X 0,Y 381.121,Z 595.57,A -85,B 0,C 180,E1 -12507.736,E2 -12507.736} C_VEL
LIN {X 0,Y 380.47,Z 606.346,A -85,B 0,C 180,E1 -12508.717,E2 -12508.717} C_VEL
LIN {X 0,Y 379.695,Z 617.531,A -85,B 0,C 180,E1 -12509.999,E2 -12509.999} C_VEL
LIN {X 0,Y 378.981,Z 626.839,A -85,B 0,C 180,E1 -12511.327,E2 -12511.327} C_VEL
LIN {X 0,Y 378.192,Z 635.823,A -85,B 0,C 180,E1 -12512.928,E2 -12512.928} C_VEL
LIN {X 0,Y 377.585,Z 643.062,A -85,B 0,C 180,E1 -12514.536,E2 -12514.536} C_VEL
LIN {X 0,Y 377.149,Z 647.983,A -85,B 0,C 180,E1 -12515.882,E2 -12515.882} C_VEL
LIN {X 0,Y 376.746,Z 652.765,A -85,B 0,C 180,E1 -12517.502,E2 -12517.502} C_VEL
LIN {X 0,Y 376.352,Z 656.467,A -85,B 0,C 180,E1 -12519.132,E2 -12519.132} C_VEL
LIN {X 0,Y 376.14,Z 659.141,A -85,B 0,C 180,E1 -12520.768,E2 -12520.768} C_VEL
LIN {X 0,Y 376.063,Z 660.409,A -85,B 0,C 180,E1 -12521.862,E2 -12521.862} C_VEL
LIN {X 0,Y 376.063,Z 661.575,A -85,B 0,C 180,E1 -12523.642,E2 -12523.642} C_VEL
LIN {X 0,Y 376.091,Z 661.712,A -85,B 0,C 180,E1 -12525.165,E2 -12525.165} C_VEL
LIN {X 0,Y 376.218,Z 661.352,A -85,B 0,C 180,E1 -12526.272,E2 -12526.272} C_VEL
LIN {X 0,Y 376.456,Z 660.125,A -85,B 0,C 180,E1 -12527.805,E2 -12527.805} C_VEL
LIN {X 0,Y 376.879,Z 657.659,A -85,B 0,C 180,E1 -12529.612,E2 -12529.612} C_VEL
LIN {X 0,Y 377.483,Z 653.942,A -85,B 0,C 180,E1 -12531.425,E2 -12531.425} C_VEL
LIN {X 0,Y 378.081,Z 649.703,A -85,B 0,C 180,E1 -12532.976,E2 -12532.976} C_VEL
LIN {X 0,Y 378.981,Z 643.034,A -85,B 0,C 180,E1 -12534.85,E2 -12534.85} C_VEL
LIN {X 0,Y 379.86,Z 636.248,A -85,B 0,C 180,E1 -12536.36,E2 -12536.36} C_VEL
LIN {X 0,Y 380.807,Z 628.625,A -85,B 0,C 180,E1 -12537.744,E2 -12537.744} C_VEL
LIN {X 0,Y 381.85,Z 618.788,A -85,B 0,C 180,E1 -12539.191,E2 -12539.191} C_VEL
LIN {X 0,Y 382.734,Z 609.07,A -85,B 0,C 180,E1 -12540.341,E2 -12540.341} C_VEL
LIN {X 0,Y 383.494,Z 599.961,A -85,B 0,C 180,E1 -12541.22,E2 -12541.22} C_VEL
LIN {X 0,Y 381.165,Z 592.074,A -85,B 0,C 180,E1 -12542.058,E2 -12542.058} C_VEL
LIN {X 0,Y 379.385,Z 589.247,A -85,B 0,C 180,E1 -12542.396,E2 -12542.396} C_VEL
LIN {X 0,Y 370.605,Z 581.959,A -85,B 0,C 180,E1 -12543.52,E2 -12543.52} C_VEL
LIN {X 0,Y 369.021,Z 578.891,A -85,B 0,C 180,E1 -12543.816,E2 -12543.816} C_VEL
LIN {X 0,Y 368.923,Z 578.527,A -85,B 0,C 180,E1 -12543.893,E2 -12543.893} C_VEL
LIN {X 0,Y 368.981,Z 578.62,A -85,B 0,C 180,E1 -12546.822,E2 -12546.822} C_VEL
LIN {X 0,Y 370.045,Z 584.746,A -85,B 0,C 180,E1 -12549.51,E2 -12549.51} C_VEL
LIN {X 0,Y 370.454,Z 589.475,A -85,B 0,C 180,E1 -12551.604,E2 -12551.604} C_VEL
LIN {X 0,Y 370.282,Z 596.558,A -85,B 0,C 180,E1 -12554.607,E2 -12554.607} C_VEL
LIN {X 0,Y 369.969,Z 604.092,A -85,B 0,C 180,E1 -12557.802,E2 -12557.802} C_VEL
LIN {X 0,Y 369.631,Z 613.737,A -85,B 0,C 180,E1 -12561.867,E2 -12561.867} C_VEL
LIN {X 0,Y 369.312,Z 623.25,A -85,B 0,C 180,E1 -12565.849,E2 -12565.849} C_VEL
LIN {X 0,Y 369.078,Z 628.527,A -85,B 0,C 180,E1 -12568.056,E2 -12568.056} C_VEL
LIN {X 0,Y 372.096,Z 643.622,A -85,B 0,C 180,E1 -12568.773,E2 -12568.773} C_VEL
LIN {X 0,Y 373.678,Z 652.419,A -85,B 0,C 180,E1 -12569.311,E2 -12569.311} C_VEL
LIN {X 0,Y 373.027,Z 665.228,A -85,B 0,C 180,E1 -12570.175,E2 -12570.175} C_VEL
LIN {X 0,Y 372.125,Z 677.091,A -85,B 0,C 180,E1 -12571.211,E2 -12571.211} C_VEL
LIN {X 0,Y 371.266,Z 687.663,A -85,B 0,C 180,E1 -12572.369,E2 -12572.369} C_VEL
LIN {X 0,Y 370.554,Z 696.395,A -85,B 0,C 180,E1 -12573.532,E2 -12573.532} C_VEL
LIN {X 0,Y 369.758,Z 705.423,A -85,B 0,C 180,E1 -12574.982,E2 -12574.982} C_VEL
LIN {X 0,Y 368.958,Z 714.085,A -85,B 0,C 180,E1 -12576.719,E2 -12576.719} C_VEL
LIN {X 0,Y 368.45,Z 721.007,A -85,B 0,C 180,E1 -12578.458,E2 -12578.458} C_VEL
LIN {X 0,Y 368.082,Z 725.584,A -85,B 0,C 180,E1 -12579.899,E2 -12579.899} C_VEL
LIN {X 0,Y 367.802,Z 729.897,A -85,B 0,C 180,E1 -12581.623,E2 -12581.623} C_VEL
LIN {X 0,Y 367.598,Z 733.019,A -85,B 0,C 180,E1 -12583.335,E2 -12583.335} C_VEL
LIN {X 0,Y 367.458,Z 734.484,A -85,B 0,C 180,E1 -12584.469,E2 -12584.469} C_VEL
LIN {X 0,Y 367.443,Z 735.528,A -85,B 0,C 180,E1 -12585.603,E2 -12585.603} C_VEL
LIN {X 0,Y 367.507,Z 736.231,A -85,B 0,C 180,E1 -12587.231,E2 -12587.231} C_VEL
LIN {X 0,Y 367.562,Z 735.992,A -85,B 0,C 180,E1 -12588.977,E2 -12588.977} C_VEL
LIN {X 0,Y 367.635,Z 735.31,A -85,B 0,C 180,E1 -12590.093,E2 -12590.093} C_VEL
LIN {X 0,Y 367.794,Z 734.161,A -85,B 0,C 180,E1 -12591.207,E2 -12591.207} C_VEL
LIN {X 0,Y 368.154,Z 731.333,A -85,B 0,C 180,E1 -12593.047,E2 -12593.047} C_VEL
LIN {X 0,Y 368.614,Z 726.771,A -85,B 0,C 180,E1 -12595.079,E2 -12595.079} C_VEL
LIN {X 0,Y 369.188,Z 721.767,A -85,B 0,C 180,E1 -12596.727,E2 -12596.727} C_VEL
LIN {X 0,Y 370.118,Z 714.302,A -85,B 0,C 180,E1 -12598.64,E2 -12598.64} C_VEL
LIN {X 0,Y 371.127,Z 706.217,A -85,B 0,C 180,E1 -12600.272,E2 -12600.272} C_VEL
LIN {X 0,Y 372.138,Z 697.974,A -85,B 0,C 180,E1 -12601.624,E2 -12601.624} C_VEL
LIN {X 0,Y 373.439,Z 686.858,A -85,B 0,C 180,E1 -12603.107,E2 -12603.107} C_VEL
LIN {X 0,Y 374.647,Z 675.519,A -85,B 0,C 180,E1 -12604.304,E2 -12604.304} C_VEL
LIN {X 0,Y 375.683,Z 664.063,A -85,B 0,C 180,E1 -12605.27,E2 -12605.27} C_VEL
LIN {X 0,Y 376.253,Z 655.829,A -85,B 0,C 180,E1 -12605.829,E2 -12605.829} C_VEL
LIN {X 0,Y 373.742,Z 643.568,A -85,B 0,C 180,E1 -12606.733,E2 -12606.733} C_VEL
LIN {X 0,Y 371.021,Z 634.283,A -85,B 0,C 180,E1 -12607.357,E2 -12607.357} C_VEL
LIN {X 0,Y 370.171,Z 631.726,A -85,B 0,C 180,E1 -12607.535,E2 -12607.535} C_VEL
LIN {X 0,Y 370.612,Z 625.023,A -85,B 0,C 180,E1 -12610.379,E2 -12610.379} C_VEL
LIN {X 0,Y 371.077,Z 615.955,A -85,B 0,C 180,E1 -12614.254,E2 -12614.254} C_VEL
LIN {X 0,Y 371.537,Z 608.12,A -85,B 0,C 180,E1 -12617.618,E2 -12617.618} C_VEL
LIN {X 0,Y 372.088,Z 600.142,A -85,B 0,C 180,E1 -12621.031,E2 -12621.031} C_VEL
LIN {X 0,Y 372.267,Z 594.678,A -85,B 0,C 180,E1 -12623.357,E2 -12623.357} C_VEL
LIN {X 0,Y 371.922,Z 591.26,A -85,B 0,C 180,E1 -12624.906,E2 -12624.906} C_VEL
LIN {X 0,Y 370.772,Z 585.566,A -85,B 0,C 180,E1 -12627.671,E2 -12627.671} C_VEL
LIN {X 0,Y 369.497,Z 580.579,A -85,B 0,C 180,E1 -12630.268,E2 -12630.268} C_VEL
LIN {X 0,Y 368.914,Z 578.533,A -85,B 0,C 180,E1 -12631.433,E2 -12631.433} C_VEL
LIN {X 0,Y 368.924,Z 578.532,A -85,B 0,C 180,E1 -12635.003,E2 -12635.003} C_VEL
LIN {X 0,Y 368.908,Z 578.532,A -85,B 0,C 180,E1 -12638.642,E2 -12638.642} C_VEL
LIN {X 0,Y 368.938,Z 578.523,A -85,B 0,C 180,E1 -12642.021,E2 -12642.021} C_VEL
LIN {X 0,Y 368.996,Z 578.689,A -85,B 0,C 180,E1 -12643.116,E2 -12643.116} C_VEL
LIN {X 0,Y 370.438,Z 585.521,A -85,B 0,C 180,E1 -12646.133,E2 -12646.133} C_VEL
LIN {X 0,Y 372.443,Z 595.257,A -85,B 0,C 180,E1 -12650.092,E2 -12650.092} C_VEL
LIN {X 0,Y 373.315,Z 600.971,A -85,B 0,C 180,E1 -12652.25,E2 -12652.25} C_VEL
LIN {X 0,Y 372.851,Z 606.761,A -85,B 0,C 180,E1 -12654.246,E2 -12654.246} C_VEL
LIN {X 0,Y 371.528,Z 618.181,A -85,B 0,C 180,E1 -12658.019,E2 -12658.019} C_VEL
LIN {X 0,Y 370.434,Z 629.666,A -85,B 0,C 180,E1 -12661.687,E2 -12661.687} C_VEL
LIN {X 0,Y 369.495,Z 642.5,A -85,B 0,C 180,E1 -12665.674,E2 -12665.674} C_VEL
LIN {X 0,Y 368.789,Z 653.522,A -85,B 0,C 180,E1 -12669.035,E2 -12669.035} C_VEL
LIN {X 0,Y 369.448,Z 658.159,A -85,B 0,C 180,E1 -12669.433,E2 -12669.433} C_VEL
LIN {X 0,Y 372,Z 672.593,A -85,B 0,C 180,E1 -12670.108,E2 -12670.108} C_VEL
LIN {X 0,Y 373.162,Z 684.991,A -85,B 0,C 180,E1 -12670.741,E2 -12670.741} C_VEL
LIN {X 0,Y 373.499,Z 698.874,A -85,B 0,C 180,E1 -12671.63,E2 -12671.63} C_VEL
LIN {X 0,Y 373.576,Z 707.835,A -85,B 0,C 180,E1 -12672.342,E2 -12672.342} C_VEL
LIN {X 0,Y 372.376,Z 719.74,A -85,B 0,C 180,E1 -12673.415,E2 -12673.415} C_VEL
LIN {X 0,Y 371.192,Z 730.511,A -85,B 0,C 180,E1 -12674.63,E2 -12674.63} C_VEL
LIN {X 0,Y 370.128,Z 740.298,A -85,B 0,C 180,E1 -12675.991,E2 -12675.991} C_VEL
LIN {X 0,Y 369.385,Z 748.407,A -85,B 0,C 180,E1 -12677.362,E2 -12677.362} C_VEL
LIN {X 0,Y 368.532,Z 756.429,A -85,B 0,C 180,E1 -12679.007,E2 -12679.007} C_VEL
LIN {X 0,Y 368.095,Z 762.895,A -85,B 0,C 180,E1 -12680.661,E2 -12680.661} C_VEL
LIN {X 0,Y 367.793,Z 768.079,A -85,B 0,C 180,E1 -12682.314,E2 -12682.314} C_VEL
LIN {X 0,Y 367.66,Z 771.601,A -85,B 0,C 180,E1 -12683.727,E2 -12683.727} C_VEL
LIN {X 0,Y 367.615,Z 775.046,A -85,B 0,C 180,E1 -12685.615,E2 -12685.615} C_VEL
LIN {X 0,Y 367.577,Z 776.454,A -85,B 0,C 180,E1 -12686.713,E2 -12686.713} C_VEL
LIN {X 0,Y 367.701,Z 777.456,A -85,B 0,C 180,E1 -12687.81,E2 -12687.81} C_VEL
LIN {X 0,Y 367.7,Z 777.983,A -85,B 0,C 180,E1 -12688.906,E2 -12688.906} C_VEL
LIN {X 0,Y 367.715,Z 778.091,A -85,B 0,C 180,E1 -12690.001,E2 -12690.001} C_VEL
LIN {X 0,Y 367.71,Z 777.789,A -85,B 0,C 180,E1 -12691.096,E2 -12691.096} C_VEL
LIN {X 0,Y 367.723,Z 777.053,A -85,B 0,C 180,E1 -12692.192,E2 -12692.192} C_VEL
LIN {X 0,Y 367.6,Z 775.843,A -85,B 0,C 180,E1 -12693.289,E2 -12693.289} C_VEL
LIN {X 0,Y 367.692,Z 773.227,A -85,B 0,C 180,E1 -12694.935,E2 -12694.935} C_VEL
LIN {X 0,Y 367.684,Z 769.515,A -85,B 0,C 180,E1 -12696.586,E2 -12696.586} C_VEL
LIN {X 0,Y 367.865,Z 764.629,A -85,B 0,C 180,E1 -12698.239,E2 -12698.239} C_VEL
LIN {X 0,Y 368.19,Z 758.424,A -85,B 0,C 180,E1 -12699.893,E2 -12699.893} C_VEL
LIN {X 0,Y 368.705,Z 750.643,A -85,B 0,C 180,E1 -12701.546,E2 -12701.546} C_VEL
LIN {X 0,Y 369.482,Z 740.887,A -85,B 0,C 180,E1 -12703.195,E2 -12703.195} C_VEL
LIN {X 0,Y 370.068,Z 732.954,A -85,B 0,C 180,E1 -12704.294,E2 -12704.294} C_VEL
LIN {X 0,Y 370.933,Z 722.196,A -85,B 0,C 180,E1 -12705.524,E2 -12705.524} C_VEL
LIN {X 0,Y 371.931,Z 710.094,A -85,B 0,C 180,E1 -12706.608,E2 -12706.608} C_VEL
LIN {X 0,Y 372.183,Z 702.636,A -85,B 0,C 180,E1 -12707.161,E2 -12707.161} C_VEL
LIN {X 0,Y 371.513,Z 691.016,A -85,B 0,C 180,E1 -12707.886,E2 -12707.886} C_VEL
LIN {X 0,Y 370.496,Z 677.497,A -85,B 0,C 180,E1 -12708.513,E2 -12708.513} C_VEL
LIN {X 0,Y 368.613,Z 658.997,A -85,B 0,C 180,E1 -12709.13,E2 -12709.13} C_VEL
LIN {X 0,Y 368.485,Z 656.897,A -85,B 0,C 180,E1 -12709.282,E2 -12709.282} C_VEL
LIN {X 0,Y 369.007,Z 644.385,A -85,B 0,C 180,E1 -12712.983,E2 -12712.983} C_VEL
LIN {X 0,Y 369.736,Z 632.002,A -85,B 0,C 180,E1 -12716.698,E2 -12716.698} C_VEL
LIN {X 0,Y 370.566,Z 620.557,A -85,B 0,C 180,E1 -12720.172,E2 -12720.172} C_VEL
LIN {X 0,Y 371.512,Z 609.359,A -85,B 0,C 180,E1 -12723.657,E2 -12723.657} C_VEL
LIN {X 0,Y 372.412,Z 599.431,A -85,B 0,C 180,E1 -12726.812,E2 -12726.812} C_VEL
LIN {X 0,Y 372.243,Z 595.846,A -85,B 0,C 180,E1 -12728.008,E2 -12728.008} C_VEL
LIN {X 0,Y 370.541,Z 586.726,A -85,B 0,C 180,E1 -12731.229,E2 -12731.229} C_VEL
LIN {X 0,Y 368.904,Z 578.535,A -85,B 0,C 180,E1 -12734.352,E2 -12734.352} C_VEL
LIN {X 0,Y 368.888,Z 578.537,A -85,B 0,C 180,E1 -12738.178,E2 -12738.178} C_VEL
LIN {X 0,Y 368.915,Z 578.529,A -85,B 0,C 180,E1 -12741.359,E2 -12741.359} C_VEL
LIN {X 0,Y 368.942,Z 578.525,A -85,B 0,C 180,E1 -12745.147,E2 -12745.147} C_VEL
LIN {X 0,Y 368.934,Z 578.527,A -85,B 0,C 180,E1 -12749.046,E2 -12749.046} C_VEL
LIN {X 0,Y 368.968,Z 578.524,A -85,B 0,C 180,E1 -12752.796,E2 -12752.796} C_VEL
LIN {X 0,Y 368.95,Z 578.529,A -85,B 0,C 180,E1 -12756.113,E2 -12756.113} C_VEL
LIN {X 0,Y 368.942,Z 578.528,A -85,B 0,C 180,E1 -12759.947,E2 -12759.947} C_VEL
LIN {X 0,Y 368.98,Z 578.52,A -85,B 0,C 180,E1 -12763.398,E2 -12763.398} C_VEL
LIN {X 0,Y 369.062,Z 578.513,A -85,B 0,C 180,E1 -12766.79,E2 -12766.79} C_VEL
LIN {X 0,Y 369.072,Z 578.513,A -85,B 0,C 180,E1 -12770.131,E2 -12770.131} C_VEL
LIN {X 0,Y 369.193,Z 578.499,A -85,B 0,C 180,E1 -12772.342,E2 -12772.342} C_VEL
LIN {X 0,Y 369.148,Z 578.505,A -85,B 0,C 180,E1 -12774.537,E2 -12774.537} C_VEL
LIN {X 0,Y 369.32,Z 578.479,A -85,B 0,C 180,E1 -12777.818,E2 -12777.818} C_VEL
LIN {X 0,Y 369.462,Z 578.463,A -85,B 0,C 180,E1 -12780,E2 -12780} C_VEL
LIN {X 0,Y 369.32,Z 578.482,A -85,B 0,C 180,E1 -12782.181,E2 -12782.181} C_VEL
LIN {X 0,Y 369.208,Z 578.496,A -85,B 0,C 180,E1 -12786.611,E2 -12786.611} C_VEL
LIN {X 0,Y 369.141,Z 578.503,A -85,B 0,C 180,E1 -12788.76,E2 -12788.76} C_VEL
LIN {X 0,Y 369.008,Z 578.52,A -85,B 0,C 180,E1 -12792.093,E2 -12792.093} C_VEL
LIN {X 0,Y 369.001,Z 578.518,A -85,B 0,C 180,E1 -12795.464,E2 -12795.464} C_VEL
LIN {X 0,Y 368.985,Z 578.522,A -85,B 0,C 180,E1 -12798.892,E2 -12798.892} C_VEL
LIN {X 0,Y 368.935,Z 578.532,A -85,B 0,C 180,E1 -12802.394,E2 -12802.394} C_VEL
LIN {X 0,Y 369.002,Z 578.52,A -85,B 0,C 180,E1 -12805.979,E2 -12805.979} C_VEL
LIN {X 0,Y 368.963,Z 578.526,A -85,B 0,C 180,E1 -12808.811,E2 -12808.811} C_VEL
LIN {X 0,Y 368.9,Z 578.535,A -85,B 0,C 180,E1 -12812.237,E2 -12812.237} C_VEL
LIN {X 0,Y 368.931,Z 578.528,A -85,B 0,C 180,E1 -12815.001,E2 -12815.001} C_VEL
LIN {X 0,Y 368.912,Z 578.534,A -85,B 0,C 180,E1 -12818.64,E2 -12818.64} C_VEL
LIN {X 0,Y 368.883,Z 578.534,A -85,B 0,C 180,E1 -12822.009,E2 -12822.009} C_VEL
LIN {X 0,Y 368.888,Z 578.533,A -85,B 0,C 180,E1 -12825.176,E2 -12825.176} C_VEL
LIN {X 0,Y 368.885,Z 578.535,A -85,B 0,C 180,E1 -12828.177,E2 -12828.177} C_VEL
LIN {X 0,Y 368.91,Z 578.529,A -85,B 0,C 180,E1 -12831.359,E2 -12831.359} C_VEL
LIN {X 0,Y 368.937,Z 578.527,A -85,B 0,C 180,E1 -12835.146,E2 -12835.146} C_VEL
LIN {X 0,Y 368.929,Z 578.529,A -85,B 0,C 180,E1 -12839.046,E2 -12839.046} C_VEL
LIN {X 0,Y 368.963,Z 578.526,A -85,B 0,C 180,E1 -12842.796,E2 -12842.796} C_VEL
LIN {X 0,Y 368.945,Z 578.527,A -85,B 0,C 180,E1 -12846.112,E2 -12846.112} C_VEL
LIN {X 0,Y 368.936,Z 578.527,A -85,B 0,C 180,E1 -12849.946,E2 -12849.946} C_VEL
LIN {X 0,Y 368.975,Z 578.521,A -85,B 0,C 180,E1 -12853.398,E2 -12853.398} C_VEL
LIN {X 0,Y 369.059,Z 578.515,A -85,B 0,C 180,E1 -12856.789,E2 -12856.789} C_VEL
LIN {X 0,Y 369.071,Z 578.511,A -85,B 0,C 180,E1 -12860.131,E2 -12860.131} C_VEL
LIN {X 0,Y 369.188,Z 578.499,A -85,B 0,C 180,E1 -12862.341,E2 -12862.341} C_VEL
LIN {X 0,Y 369.145,Z 578.505,A -85,B 0,C 180,E1 -12864.537,E2 -12864.537} C_VEL
LIN {X 0,Y 369.083,Z 578.654,A -85,B 0,C 180,E1 -12866.007,E2 -12866.007} C_VEL
LIN {X 0,Y 372.517,Z 589.919,A -85,B 0,C 180,E1 -12866.887,E2 -12866.887} C_VEL
LIN {X 0,Y 374.239,Z 597.169,A -85,B 0,C 180,E1 -12867.543,E2 -12867.543} C_VEL
LIN {X 0,Y 373.508,Z 608.864,A -85,B 0,C 180,E1 -12868.651,E2 -12868.651} C_VEL
LIN {X 0,Y 372.824,Z 618.36,A -85,B 0,C 180,E1 -12869.774,E2 -12869.774} C_VEL
LIN {X 0,Y 372.107,Z 627.414,A -85,B 0,C 180,E1 -12871.081,E2 -12871.081} C_VEL
LIN {X 0,Y 371.389,Z 635.148,A -85,B 0,C 180,E1 -12872.439,E2 -12872.439} C_VEL
LIN {X 0,Y 370.758,Z 642.681,A -85,B 0,C 180,E1 -12874.075,E2 -12874.075} C_VEL
LIN {X 0,Y 370.103,Z 649.665,A -85,B 0,C 180,E1 -12875.994,E2 -12875.994} C_VEL
LIN {X 0,Y 369.694,Z 654.309,A -85,B 0,C 180,E1 -12877.646,E2 -12877.646} C_VEL
LIN {X 0,Y 369.301,Z 657.882,A -85,B 0,C 180,E1 -12879.308,E2 -12879.308} C_VEL
LIN {X 0,Y 369.112,Z 660.43,A -85,B 0,C 180,E1 -12880.975,E2 -12880.975} C_VEL
LIN {X 0,Y 369.028,Z 661.618,A -85,B 0,C 180,E1 -12882.091,E2 -12882.091} C_VEL
LIN {X 0,Y 369.047,Z 662.621,A -85,B 0,C 180,E1 -12883.78,E2 -12883.78} C_VEL
LIN {X 0,Y 369.102,Z 662.708,A -85,B 0,C 180,E1 -12885.459,E2 -12885.459} C_VEL
LIN {X 0,Y 369.232,Z 662.239,A -85,B 0,C 180,E1 -12886.588,E2 -12886.588} C_VEL
LIN {X 0,Y 369.5,Z 661.075,A -85,B 0,C 180,E1 -12888.009,E2 -12888.009} C_VEL
LIN {X 0,Y 370.005,Z 658.308,A -85,B 0,C 180,E1 -12889.991,E2 -12889.991} C_VEL
LIN {X 0,Y 370.607,Z 654.8,A -85,B 0,C 180,E1 -12891.689,E2 -12891.689} C_VEL
LIN {X 0,Y 371.307,Z 650.039,A -85,B 0,C 180,E1 -12893.42,E2 -12893.42} C_VEL
LIN {X 0,Y 372.212,Z 643.72,A -85,B 0,C 180,E1 -12895.197,E2 -12895.197} C_VEL
LIN {X 0,Y 373.287,Z 636.225,A -85,B 0,C 180,E1 -12896.861,E2 -12896.861} C_VEL
LIN {X 0,Y 374.301,Z 628.166,A -85,B 0,C 180,E1 -12898.3,E2 -12898.3} C_VEL
LIN {X 0,Y 375.357,Z 618.165,A -85,B 0,C 180,E1 -12899.746,E2 -12899.746} C_VEL
LIN {X 0,Y 376.416,Z 607.536,A -85,B 0,C 180,E1 -12900.971,E2 -12900.971} C_VEL
LIN {X 0,Y 376.88,Z 602.318,A -85,B 0,C 180,E1 -12901.474,E2 -12901.474} C_VEL
LIN {X 0,Y 374.906,Z 595.13,A -85,B 0,C 180,E1 -12902.264,E2 -12902.264} C_VEL
LIN {X 0,Y 371.191,Z 584.776,A -85,B 0,C 180,E1 -12903.302,E2 -12903.302} C_VEL
LIN {X 0,Y 369.021,Z 578.891,A -85,B 0,C 180,E1 -12903.816,E2 -12903.816} C_VEL
LIN {X 0,Y 368.415,Z 578.59,A -85,B 0,C 180,E1 -12903.998,E2 -12903.998} C_VEL
LIN {X 0,Y 364.255,Z 579.287,A -85,B 0,C 180,E1 -12905.378,E2 -12905.378} C_VEL
LIN {X 0,Y 362.475,Z 579.626,A -85,B 0,C 180,E1 -12906.279,E2 -12906.279} C_VEL
LIN {X 0,Y 362.076,Z 580.414,A -85,B 0,C 180,E1 -12906.963,E2 -12906.963} C_VEL
LIN {X 0,Y 363.143,Z 586.498,A -85,B 0,C 180,E1 -12909.69,E2 -12909.69} C_VEL
LIN {X 0,Y 363.466,Z 591.39,A -85,B 0,C 180,E1 -12911.841,E2 -12911.841} C_VEL
LIN {X 0,Y 363.248,Z 598.912,A -85,B 0,C 180,E1 -12915.066,E2 -12915.066} C_VEL
LIN {X 0,Y 362.923,Z 606.029,A -85,B 0,C 180,E1 -12918.089,E2 -12918.089} C_VEL
LIN {X 0,Y 362.624,Z 614.433,A -85,B 0,C 180,E1 -12921.671,E2 -12921.671} C_VEL
LIN {X 0,Y 362.302,Z 624.101,A -85,B 0,C 180,E1 -12925.768,E2 -12925.768} C_VEL
LIN {X 0,Y 362.1,Z 628.86,A -85,B 0,C 180,E1 -12927.765,E2 -12927.765} C_VEL
LIN {X 0,Y 365.112,Z 644.136,A -85,B 0,C 180,E1 -12928.511,E2 -12928.511} C_VEL
LIN {X 0,Y 366.79,Z 653.964,A -85,B 0,C 180,E1 -12929.132,E2 -12929.132} C_VEL
LIN {X 0,Y 366.117,Z 665.595,A -85,B 0,C 180,E1 -12929.94,E2 -12929.94} C_VEL
LIN {X 0,Y 365.235,Z 676.826,A -85,B 0,C 180,E1 -12930.931,E2 -12930.931} C_VEL
LIN {X 0,Y 364.252,Z 688.714,A -85,B 0,C 180,E1 -12932.26,E2 -12932.26} C_VEL
LIN {X 0,Y 363.426,Z 698.323,A -85,B 0,C 180,E1 -12933.591,E2 -12933.591} C_VEL
LIN {X 0,Y 362.641,Z 706.905,A -85,B 0,C 180,E1 -12935.046,E2 -12935.046} C_VEL
LIN {X 0,Y 361.844,Z 715.501,A -85,B 0,C 180,E1 -12936.84,E2 -12936.84} C_VEL
LIN {X 0,Y 361.418,Z 721.186,A -85,B 0,C 180,E1 -12938.318,E2 -12938.318} C_VEL
LIN {X 0,Y 360.96,Z 726.625,A -85,B 0,C 180,E1 -12940.079,E2 -12940.079} C_VEL
LIN {X 0,Y 360.696,Z 730.766,A -85,B 0,C 180,E1 -12941.836,E2 -12941.836} C_VEL
LIN {X 0,Y 360.548,Z 732.882,A -85,B 0,C 180,E1 -12942.999,E2 -12942.999} C_VEL
LIN {X 0,Y 360.407,Z 734.532,A -85,B 0,C 180,E1 -12944.157,E2 -12944.157} C_VEL
LIN {X 0,Y 360.348,Z 735.68,A -85,B 0,C 180,E1 -12945.313,E2 -12945.313} C_VEL
LIN {X 0,Y 360.41,Z 736.625,A -85,B 0,C 180,E1 -12947.155,E2 -12947.155} C_VEL
LIN {X 0,Y 360.465,Z 736.546,A -85,B 0,C 180,E1 -12948.757,E2 -12948.757} C_VEL
LIN {X 0,Y 360.532,Z 735.981,A -85,B 0,C 180,E1 -12949.896,E2 -12949.896} C_VEL
LIN {X 0,Y 360.689,Z 735.009,A -85,B 0,C 180,E1 -12951.033,E2 -12951.033} C_VEL
LIN {X 0,Y 361.098,Z 732.211,A -85,B 0,C 180,E1 -12953.016,E2 -12953.016} C_VEL
LIN {X 0,Y 361.557,Z 728.078,A -85,B 0,C 180,E1 -12954.982,E2 -12954.982} C_VEL
LIN {X 0,Y 362.13,Z 723.332,A -85,B 0,C 180,E1 -12956.663,E2 -12956.663} C_VEL
LIN {X 0,Y 362.918,Z 717.338,A -85,B 0,C 180,E1 -12958.336,E2 -12958.336} C_VEL
LIN {X 0,Y 363.932,Z 709.859,A -85,B 0,C 180,E1 -12960,E2 -12960} C_VEL
LIN {X 0,Y 365.164,Z 700.663,A -85,B 0,C 180,E1 -12961.655,E2 -12961.655} C_VEL
LIN {X 0,Y 366.33,Z 691.491,A -85,B 0,C 180,E1 -12962.987,E2 -12962.987} C_VEL
LIN {X 0,Y 367.597,Z 680.75,A -85,B 0,C 180,E1 -12964.249,E2 -12964.249} C_VEL
LIN {X 0,Y 368.758,Z 669.31,A -85,B 0,C 180,E1 -12965.332,E2 -12965.332} C_VEL
LIN {X 0,Y 369.702,Z 657.174,A -85,B 0,C 180,E1 -12966.228,E2 -12966.228} C_VEL
LIN {X 0,Y 367.361,Z 645.207,A -85,B 0,C 180,E1 -12967.164,E2 -12967.164} C_VEL
LIN {X 0,Y 364.246,Z 634.908,A -85,B 0,C 180,E1 -12967.902,E2 -12967.902} C_VEL
LIN {X 0,Y 363.391,Z 632.23,A -85,B 0,C 180,E1 -12968.096,E2 -12968.096} C_VEL
LIN {X 0,Y 363.828,Z 625.211,A -85,B 0,C 180,E1 -12971.138,E2 -12971.138} C_VEL
LIN {X 0,Y 364.277,Z 617.406,A -85,B 0,C 180,E1 -12974.526,E2 -12974.526} C_VEL
LIN {X 0,Y 364.823,Z 609.62,A -85,B 0,C 180,E1 -12977.953,E2 -12977.953} C_VEL
LIN {X 0,Y 365.415,Z 601.59,A -85,B 0,C 180,E1 -12981.434,E2 -12981.434} C_VEL
LIN {X 0,Y 365.609,Z 596.306,A -85,B 0,C 180,E1 -12983.809,E2 -12983.809} C_VEL
LIN {X 0,Y 364.832,Z 591.115,A -85,B 0,C 180,E1 -12986.3,E2 -12986.3} C_VEL
LIN {X 0,Y 363.729,Z 586.184,A -85,B 0,C 180,E1 -12988.885,E2 -12988.885} C_VEL
LIN {X 0,Y 362.466,Z 581.459,A -85,B 0,C 180,E1 -12991.569,E2 -12991.569} C_VEL
LIN {X 0,Y 361.843,Z 579.414,A -85,B 0,C 180,E1 -12992.946,E2 -12992.946} C_VEL
LIN {X 0,Y 361.863,Z 579.41,A -85,B 0,C 180,E1 -12995.638,E2 -12995.638} C_VEL
LIN {X 0,Y 361.87,Z 579.41,A -85,B 0,C 180,E1 -12999.029,E2 -12999.029} C_VEL
LIN {X 0,Y 361.931,Z 579.492,A -85,B 0,C 180,E1 -13002.526,E2 -13002.526} C_VEL
LIN {X 0,Y 363.505,Z 586.907,A -85,B 0,C 180,E1 -13005.893,E2 -13005.893} C_VEL
LIN {X 0,Y 365.408,Z 596.209,A -85,B 0,C 180,E1 -13009.765,E2 -13009.765} C_VEL
LIN {X 0,Y 366.388,Z 602.334,A -85,B 0,C 180,E1 -13012.136,E2 -13012.136} C_VEL
LIN {X 0,Y 366.065,Z 606.856,A -85,B 0,C 180,E1 -13013.741,E2 -13013.741} C_VEL
LIN {X 0,Y 364.733,Z 617.49,A -85,B 0,C 180,E1 -13017.35,E2 -13017.35} C_VEL
LIN {X 0,Y 363.53,Z 628.938,A -85,B 0,C 180,E1 -13021.099,E2 -13021.099} C_VEL
LIN {X 0,Y 362.586,Z 640.373,A -85,B 0,C 180,E1 -13024.76,E2 -13024.76} C_VEL
LIN {X 0,Y 361.85,Z 651.636,A -85,B 0,C 180,E1 -13028.271,E2 -13028.271} C_VEL
LIN {X 0,Y 362.556,Z 657.447,A -85,B 0,C 180,E1 -13028.844,E2 -13028.844} C_VEL
LIN {X 0,Y 365.195,Z 670.57,A -85,B 0,C 180,E1 -13029.512,E2 -13029.512} C_VEL
LIN {X 0,Y 366.462,Z 683.056,A -85,B 0,C 180,E1 -13030.172,E2 -13030.172} C_VEL
LIN {X 0,Y 366.821,Z 696.036,A -85,B 0,C 180,E1 -13030.993,E2 -13030.993} C_VEL
LIN {X 0,Y 366.87,Z 708.662,A -85,B 0,C 180,E1 -13032.008,E2 -13032.008} C_VEL
LIN {X 0,Y 365.616,Z 720.243,A -85,B 0,C 180,E1 -13033.099,E2 -13033.099} C_VEL
LIN {X 0,Y 364.358,Z 730.742,A -85,B 0,C 180,E1 -13034.334,E2 -13034.334} C_VEL
LIN {X 0,Y 363.236,Z 740.378,A -85,B 0,C 180,E1 -13035.719,E2 -13035.719} C_VEL
LIN {X 0,Y 362.423,Z 748.407,A -85,B 0,C 180,E1 -13037.116,E2 -13037.116} C_VEL
LIN {X 0,Y 361.53,Z 756.325,A -85,B 0,C 180,E1 -13038.792,E2 -13038.792} C_VEL
LIN {X 0,Y 361.039,Z 762.723,A -85,B 0,C 180,E1 -13040.477,E2 -13040.477} C_VEL
LIN {X 0,Y 360.723,Z 767.836,A -85,B 0,C 180,E1 -13042.163,E2 -13042.163} C_VEL
LIN {X 0,Y 360.565,Z 771.625,A -85,B 0,C 180,E1 -13043.763,E2 -13043.763} C_VEL
LIN {X 0,Y 360.539,Z 774.712,A -85,B 0,C 180,E1 -13045.529,E2 -13045.529} C_VEL
LIN {X 0,Y 360.487,Z 776.104,A -85,B 0,C 180,E1 -13046.648,E2 -13046.648} C_VEL
LIN {X 0,Y 360.599,Z 777.071,A -85,B 0,C 180,E1 -13047.767,E2 -13047.767} C_VEL
LIN {X 0,Y 360.63,Z 777.57,A -85,B 0,C 180,E1 -13048.884,E2 -13048.884} C_VEL
LIN {X 0,Y 360.642,Z 777.659,A -85,B 0,C 180,E1 -13050.001,E2 -13050.001} C_VEL
LIN {X 0,Y 360.639,Z 777.336,A -85,B 0,C 180,E1 -13051.118,E2 -13051.118} C_VEL
LIN {X 0,Y 360.654,Z 776.551,A -85,B 0,C 180,E1 -13052.235,E2 -13052.235} C_VEL
LIN {X 0,Y 360.511,Z 775.315,A -85,B 0,C 180,E1 -13053.354,E2 -13053.354} C_VEL
LIN {X 0,Y 360.617,Z 772.65,A -85,B 0,C 180,E1 -13055.032,E2 -13055.032} C_VEL
LIN {X 0,Y 360.6,Z 768.883,A -85,B 0,C 180,E1 -13056.716,E2 -13056.716} C_VEL
LIN {X 0,Y 360.807,Z 763.941,A -85,B 0,C 180,E1 -13058.401,E2 -13058.401} C_VEL
LIN {X 0,Y 361.161,Z 757.674,A -85,B 0,C 180,E1 -13060.087,E2 -13060.087} C_VEL
LIN {X 0,Y 361.714,Z 749.781,A -85,B 0,C 180,E1 -13061.773,E2 -13061.773} C_VEL
LIN {X 0,Y 362.339,Z 741.712,A -85,B 0,C 180,E1 -13063.175,E2 -13063.175} C_VEL
LIN {X 0,Y 362.995,Z 733.469,A -85,B 0,C 180,E1 -13064.367,E2 -13064.367} C_VEL
LIN {X 0,Y 363.914,Z 722.33,A -85,B 0,C 180,E1 -13065.687,E2 -13065.687} C_VEL
LIN {X 0,Y 364.946,Z 710.386,A -85,B 0,C 180,E1 -13066.791,E2 -13066.791} C_VEL
LIN {X 0,Y 365.189,Z 703.079,A -85,B 0,C 180,E1 -13067.356,E2 -13067.356} C_VEL
LIN {X 0,Y 364.568,Z 691.033,A -85,B 0,C 180,E1 -13068.129,E2 -13068.129} C_VEL
LIN {X 0,Y 363.532,Z 677.316,A -85,B 0,C 180,E1 -13068.783,E2 -13068.783} C_VEL
LIN {X 0,Y 361.649,Z 658.604,A -85,B 0,C 180,E1 -13069.439,E2 -13069.439} C_VEL
LIN {X 0,Y 361.48,Z 655.654,A -85,B 0,C 180,E1 -13069.67,E2 -13069.67} C_VEL
LIN {X 0,Y 362.014,Z 643.215,A -85,B 0,C 180,E1 -13073.453,E2 -13073.453} C_VEL
LIN {X 0,Y 362.921,Z 629.409,A -85,B 0,C 180,E1 -13077.696,E2 -13077.696} C_VEL
LIN {X 0,Y 363.95,Z 616.193,A -85,B 0,C 180,E1 -13081.825,E2 -13081.825} C_VEL
LIN {X 0,Y 364.97,Z 605.395,A -85,B 0,C 180,E1 -13085.289,E2 -13085.289} C_VEL
LIN {X 0,Y 365.463,Z 598.443,A -85,B 0,C 180,E1 -13087.579,E2 -13087.579} C_VEL
LIN {X 0,Y 363.913,Z 589.668,A -85,B 0,C 180,E1 -13090.711,E2 -13090.711} C_VEL
LIN {X 0,Y 361.99,Z 580.091,A -85,B 0,C 180,E1 -13094.343,E2 -13094.343} C_VEL
LIN {X 0,Y 361.867,Z 579.411,A -85,B 0,C 180,E1 -13094.655,E2 -13094.655} C_VEL
LIN {X 0,Y 361.841,Z 579.413,A -85,B 0,C 180,E1 -13097.568,E2 -13097.568} C_VEL
LIN {X 0,Y 361.876,Z 579.406,A -85,B 0,C 180,E1 -13100.973,E2 -13100.973} C_VEL
LIN {X 0,Y 361.88,Z 579.408,A -85,B 0,C 180,E1 -13104.655,E2 -13104.655} C_VEL
LIN {X 0,Y 361.843,Z 579.415,A -85,B 0,C 180,E1 -13108.371,E2 -13108.371} C_VEL
LIN {X 0,Y 361.913,Z 579.406,A -85,B 0,C 180,E1 -13112.221,E2 -13112.221} C_VEL
LIN {X 0,Y 361.933,Z 579.401,A -85,B 0,C 180,E1 -13114.71,E2 -13114.71} C_VEL
LIN {X 0,Y 361.897,Z 579.408,A -85,B 0,C 180,E1 -13118.347,E2 -13118.347} C_VEL
LIN {X 0,Y 361.972,Z 579.397,A -85,B 0,C 180,E1 -13122.061,E2 -13122.061} C_VEL
LIN {X 0,Y 362.003,Z 579.393,A -85,B 0,C 180,E1 -13126.101,E2 -13126.101} C_VEL
LIN {X 0,Y 362.036,Z 579.388,A -85,B 0,C 180,E1 -13129.938,E2 -13129.938} C_VEL
LIN {X 0,Y 362.151,Z 579.375,A -85,B 0,C 180,E1 -13132.192,E2 -13132.192} C_VEL
LIN {X 0,Y 362.122,Z 579.38,A -85,B 0,C 180,E1 -13134.431,E2 -13134.431} C_VEL
LIN {X 0,Y 362.284,Z 579.355,A -85,B 0,C 180,E1 -13137.776,E2 -13137.776} C_VEL
LIN {X 0,Y 362.432,Z 579.338,A -85,B 0,C 180,E1 -13140,E2 -13140} C_VEL
LIN {X 0,Y 362.284,Z 579.359,A -85,B 0,C 180,E1 -13142.223,E2 -13142.223} C_VEL
LIN {X 0,Y 362.176,Z 579.371,A -85,B 0,C 180,E1 -13146.686,E2 -13146.686} C_VEL
LIN {X 0,Y 362.078,Z 579.382,A -85,B 0,C 180,E1 -13148.933,E2 -13148.933} C_VEL
LIN {X 0,Y 361.964,Z 579.4,A -85,B 0,C 180,E1 -13152.332,E2 -13152.332} C_VEL
LIN {X 0,Y 361.965,Z 579.399,A -85,B 0,C 180,E1 -13154.62,E2 -13154.62} C_VEL
LIN {X 0,Y 361.963,Z 579.398,A -85,B 0,C 180,E1 -13158.099,E2 -13158.099} C_VEL
LIN {X 0,Y 361.895,Z 579.403,A -85,B 0,C 180,E1 -13161.652,E2 -13161.652} C_VEL
LIN {X 0,Y 361.931,Z 579.399,A -85,B 0,C 180,E1 -13165.289,E2 -13165.289} C_VEL
LIN {X 0,Y 361.921,Z 579.4,A -85,B 0,C 180,E1 -13167.777,E2 -13167.777} C_VEL
LIN {X 0,Y 361.849,Z 579.409,A -85,B 0,C 180,E1 -13171.284,E2 -13171.284} C_VEL
LIN {X 0,Y 361.856,Z 579.412,A -85,B 0,C 180,E1 -13174.28,E2 -13174.28} C_VEL
LIN {X 0,Y 361.867,Z 579.407,A -85,B 0,C 180,E1 -13177.222,E2 -13177.222} C_VEL
LIN {X 0,Y 361.838,Z 579.413,A -85,B 0,C 180,E1 -13180.755,E2 -13180.755} C_VEL
LIN {X 0,Y 361.849,Z 579.414,A -85,B 0,C 180,E1 -13184.363,E2 -13184.363} C_VEL
LIN {X 0,Y 361.838,Z 579.41,A -85,B 0,C 180,E1 -13187.567,E2 -13187.567} C_VEL
LIN {X 0,Y 361.871,Z 579.408,A -85,B 0,C 180,E1 -13190.972,E2 -13190.972} C_VEL
LIN {X 0,Y 361.875,Z 579.41,A -85,B 0,C 180,E1 -13194.654,E2 -13194.654} C_VEL
LIN {X 0,Y 361.838,Z 579.415,A -85,B 0,C 180,E1 -13198.37,E2 -13198.37} C_VEL
LIN {X 0,Y 361.908,Z 579.404,A -85,B 0,C 180,E1 -13202.22,E2 -13202.22} C_VEL
LIN {X 0,Y 361.929,Z 579.404,A -85,B 0,C 180,E1 -13204.709,E2 -13204.709} C_VEL
LIN {X 0,Y 361.893,Z 579.407,A -85,B 0,C 180,E1 -13208.346,E2 -13208.346} C_VEL
LIN {X 0,Y 361.967,Z 579.396,A -85,B 0,C 180,E1 -13212.06,E2 -13212.06} C_VEL
LIN {X 0,Y 361.998,Z 579.392,A -85,B 0,C 180,E1 -13216.1,E2 -13216.1} C_VEL
LIN {X 0,Y 362.035,Z 579.386,A -85,B 0,C 180,E1 -13219.937,E2 -13219.937} C_VEL
LIN {X 0,Y 362.151,Z 579.374,A -85,B 0,C 180,E1 -13222.192,E2 -13222.192} C_VEL
LIN {X 0,Y 362.118,Z 579.38,A -85,B 0,C 180,E1 -13224.43,E2 -13224.43} C_VEL
LIN {X 0,Y 361.974,Z 579.393,A -85,B 0,C 180,E1 -13225.684,E2 -13225.684} C_VEL
LIN {X 0,Y 365.77,Z 591.826,A -85,B 0,C 180,E1 -13226.694,E2 -13226.694} C_VEL
LIN {X 0,Y 367.359,Z 597.984,A -85,B 0,C 180,E1 -13227.273,E2 -13227.273} C_VEL
LIN {X 0,Y 366.676,Z 609.228,A -85,B 0,C 180,E1 -13228.352,E2 -13228.352} C_VEL
LIN {X 0,Y 365.934,Z 619.281,A -85,B 0,C 180,E1 -13229.553,E2 -13229.553} C_VEL
LIN {X 0,Y 365.26,Z 627.666,A -85,B 0,C 180,E1 -13230.778,E2 -13230.778} C_VEL
LIN {X 0,Y 364.47,Z 635.794,A -85,B 0,C 180,E1 -13232.209,E2 -13232.209} C_VEL
LIN {X 0,Y 363.813,Z 643.412,A -85,B 0,C 180,E1 -13233.876,E2 -13233.876} C_VEL
LIN {X 0,Y 363.219,Z 649.546,A -85,B 0,C 180,E1 -13235.551,E2 -13235.551} C_VEL
LIN {X 0,Y 362.772,Z 654.426,A -85,B 0,C 180,E1 -13237.233,E2 -13237.233} C_VEL
LIN {X 0,Y 362.349,Z 658.218,A -85,B 0,C 180,E1 -13238.925,E2 -13238.925} C_VEL
LIN {X 0,Y 362.178,Z 660.176,A -85,B 0,C 180,E1 -13240.057,E2 -13240.057} C_VEL
LIN {X 0,Y 362.072,Z 661.707,A -85,B 0,C 180,E1 -13241.191,E2 -13241.191} C_VEL
LIN {X 0,Y 362.042,Z 663.472,A -85,B 0,C 180,E1 -13243.469,E2 -13243.469} C_VEL
LIN {X 0,Y 362.04,Z 663.786,A -85,B 0,C 180,E1 -13244.616,E2 -13244.616} C_VEL
LIN {X 0,Y 362.119,Z 663.662,A -85,B 0,C 180,E1 -13245.765,E2 -13245.765} C_VEL
LIN {X 0,Y 362.262,Z 663.116,A -85,B 0,C 180,E1 -13246.917,E2 -13246.917} C_VEL
LIN {X 0,Y 362.55,Z 662.024,A -85,B 0,C 180,E1 -13248.222,E2 -13248.222} C_VEL
LIN {X 0,Y 362.783,Z 660.797,A -85,B 0,C 180,E1 -13249.227,E2 -13249.227} C_VEL
LIN {X 0,Y 363.321,Z 657.861,A -85,B 0,C 180,E1 -13250.968,E2 -13250.968} C_VEL
LIN {X 0,Y 364.034,Z 653.795,A -85,B 0,C 180,E1 -13252.712,E2 -13252.712} C_VEL
LIN {X 0,Y 365.044,Z 647.443,A -85,B 0,C 180,E1 -13254.754,E2 -13254.754} C_VEL
LIN {X 0,Y 366.054,Z 640.39,A -85,B 0,C 180,E1 -13256.511,E2 -13256.511} C_VEL
LIN {X 0,Y 367.264,Z 631.908,A -85,B 0,C 180,E1 -13258.168,E2 -13258.168} C_VEL
LIN {X 0,Y 368.334,Z 622.992,A -85,B 0,C 180,E1 -13259.583,E2 -13259.583} C_VEL
LIN {X 0,Y 369.289,Z 613.912,A -85,B 0,C 180,E1 -13260.76,E2 -13260.76} C_VEL
LIN {X 0,Y 370.278,Z 603.966,A -85,B 0,C 180,E1 -13261.804,E2 -13261.804} C_VEL
LIN {X 0,Y 367.753,Z 595.544,A -85,B 0,C 180,E1 -13262.769,E2 -13262.769} C_VEL
LIN {X 0,Y 363.937,Z 584.744,A -85,B 0,C 180,E1 -13263.864,E2 -13263.864} C_VEL
LIN {X 0,Y 361.899,Z 579.403,A -85,B 0,C 180,E1 -13264.358,E2 -13264.358} C_VEL
LIN {X 0,Y 361.967,Z 579.55,A -85,B 0,C 180,E1 -13266.57,E2 -13266.57} C_VEL
LIN {X 0,Y 362.076,Z 580.414,A -85,B 0,C 180,E1 -13266.963,E2 -13266.963} C_VEL
LIN {X 0,Y 361.732,Z 582.482,A -85,B 0,C 180,E1 -13267.838,E2 -13267.838} C_VEL
LIN {X 0,Y 359.486,Z 586.214,A -85,B 0,C 180,E1 -13269.253,E2 -13269.253} C_VEL
LIN {X 0,Y 356.765,Z 590.735,A -85,B 0,C 180,E1 -13270.977,E2 -13270.977} C_VEL
LIN {X 0,Y 356.487,Z 592.159,A -85,B 0,C 180,E1 -13271.574,E2 -13271.574} C_VEL
LIN {X 0,Y 356.273,Z 599.48,A -85,B 0,C 180,E1 -13274.753,E2 -13274.753} C_VEL
LIN {X 0,Y 355.951,Z 606.646,A -85,B 0,C 180,E1 -13277.833,E2 -13277.833} C_VEL
LIN {X 0,Y 355.624,Z 615.205,A -85,B 0,C 180,E1 -13281.5,E2 -13281.5} C_VEL
LIN {X 0,Y 355.302,Z 623.377,A -85,B 0,C 180,E1 -13284.997,E2 -13284.997} C_VEL
LIN {X 0,Y 355.109,Z 629.279,A -85,B 0,C 180,E1 -13287.479,E2 -13287.479} C_VEL
LIN {X 0,Y 357.72,Z 642.469,A -85,B 0,C 180,E1 -13288.112,E2 -13288.112} C_VEL
LIN {X 0,Y 359.801,Z 654.049,A -85,B 0,C 180,E1 -13288.849,E2 -13288.849} C_VEL
LIN {X 0,Y 359.17,Z 666.586,A -85,B 0,C 180,E1 -13289.745,E2 -13289.745} C_VEL
LIN {X 0,Y 358.239,Z 678.009,A -85,B 0,C 180,E1 -13290.791,E2 -13290.791} C_VEL
LIN {X 0,Y 357.329,Z 688.561,A -85,B 0,C 180,E1 -13291.995,E2 -13291.995} C_VEL
LIN {X 0,Y 356.462,Z 698.277,A -85,B 0,C 180,E1 -13293.351,E2 -13293.351} C_VEL
LIN {X 0,Y 355.641,Z 707.071,A -85,B 0,C 180,E1 -13294.858,E2 -13294.858} C_VEL
LIN {X 0,Y 354.813,Z 715.61,A -85,B 0,C 180,E1 -13296.663,E2 -13296.663} C_VEL
LIN {X 0,Y 354.286,Z 722.407,A -85,B 0,C 180,E1 -13298.484,E2 -13298.484} C_VEL
LIN {X 0,Y 353.836,Z 727.636,A -85,B 0,C 180,E1 -13300.266,E2 -13300.266} C_VEL
LIN {X 0,Y 353.587,Z 731.749,A -85,B 0,C 180,E1 -13302.117,E2 -13302.117} C_VEL
LIN {X 0,Y 353.357,Z 734.483,A -85,B 0,C 180,E1 -13303.833,E2 -13303.833} C_VEL
LIN {X 0,Y 353.288,Z 735.818,A -85,B 0,C 180,E1 -13305.013,E2 -13305.013} C_VEL
LIN {X 0,Y 353.334,Z 737.015,A -85,B 0,C 180,E1 -13307.061,E2 -13307.061} C_VEL
LIN {X 0,Y 353.384,Z 737.096,A -85,B 0,C 180,E1 -13308.529,E2 -13308.529} C_VEL
LIN {X 0,Y 353.432,Z 736.647,A -85,B 0,C 180,E1 -13309.691,E2 -13309.691} C_VEL
LIN {X 0,Y 353.602,Z 735.78,A -85,B 0,C 180,E1 -13310.851,E2 -13310.851} C_VEL
LIN {X 0,Y 354.035,Z 733.076,A -85,B 0,C 180,E1 -13312.992,E2 -13312.992} C_VEL
LIN {X 0,Y 354.5,Z 729.359,A -85,B 0,C 180,E1 -13314.882,E2 -13314.882} C_VEL
LIN {X 0,Y 355.076,Z 724.853,A -85,B 0,C 180,E1 -13316.596,E2 -13316.596} C_VEL
LIN {X 0,Y 356.031,Z 718.09,A -85,B 0,C 180,E1 -13318.587,E2 -13318.587} C_VEL
LIN {X 0,Y 357.118,Z 710.714,A -85,B 0,C 180,E1 -13320.282,E2 -13320.282} C_VEL
LIN {X 0,Y 358.406,Z 701.587,A -85,B 0,C 180,E1 -13321.967,E2 -13321.967} C_VEL
LIN {X 0,Y 359.671,Z 692.241,A -85,B 0,C 180,E1 -13323.361,E2 -13323.361} C_VEL
LIN {X 0,Y 361.14,Z 680.691,A -85,B 0,C 180,E1 -13324.745,E2 -13324.745} C_VEL
LIN {X 0,Y 362.246,Z 670.549,A -85,B 0,C 180,E1 -13325.729,E2 -13325.729} C_VEL
LIN {X 0,Y 363.222,Z 658.443,A -85,B 0,C 180,E1 -13326.667,E2 -13326.667} C_VEL
LIN {X 0,Y 361.053,Z 646.965,A -85,B 0,C 180,E1 -13327.6,E2 -13327.6} C_VEL
LIN {X 0,Y 357.153,Z 634.649,A -85,B 0,C 180,E1 -13328.559,E2 -13328.559} C_VEL
LIN {X 0,Y 356.618,Z 632.73,A -85,B 0,C 180,E1 -13328.714,E2 -13328.714} C_VEL
LIN {X 0,Y 357.093,Z 625.447,A -85,B 0,C 180,E1 -13331.927,E2 -13331.927} C_VEL
LIN {X 0,Y 357.712,Z 616.336,A -85,B 0,C 180,E1 -13335.966,E2 -13335.966} C_VEL
LIN {X 0,Y 358.372,Z 607.942,A -85,B 0,C 180,E1 -13339.729,E2 -13339.729} C_VEL
LIN {X 0,Y 358.862,Z 602.188,A -85,B 0,C 180,E1 -13342.293,E2 -13342.293} C_VEL
LIN {X 0,Y 358.916,Z 597.951,A -85,B 0,C 180,E1 -13344.281,E2 -13344.281} C_VEL
LIN {X 0,Y 358.106,Z 592.932,A -85,B 0,C 180,E1 -13346.833,E2 -13346.833} C_VEL
LIN {X 0,Y 357.038,Z 588.157,A -85,B 0,C 180,E1 -13349.479,E2 -13349.479} C_VEL
LIN {X 0,Y 355.563,Z 582.716,A -85,B 0,C 180,E1 -13352.927,E2 -13352.927} C_VEL
LIN {X 0,Y 354.805,Z 580.293,A -85,B 0,C 180,E1 -13354.714,E2 -13354.714} C_VEL
LIN {X 0,Y 354.806,Z 580.291,A -85,B 0,C 180,E1 -13357.883,E2 -13357.883} C_VEL
LIN {X 0,Y 354.835,Z 580.286,A -85,B 0,C 180,E1 -13361.182,E2 -13361.182} C_VEL
LIN {X 0,Y 354.862,Z 580.353,A -85,B 0,C 180,E1 -13361.937,E2 -13361.937} C_VEL
LIN {X 0,Y 356.382,Z 587.362,A -85,B 0,C 180,E1 -13365.23,E2 -13365.23} C_VEL
LIN {X 0,Y 358.148,Z 596.071,A -85,B 0,C 180,E1 -13368.984,E2 -13368.984} C_VEL
LIN {X 0,Y 359.269,Z 602.288,A -85,B 0,C 180,E1 -13371.489,E2 -13371.489} C_VEL
LIN {X 0,Y 359.432,Z 605.475,A -85,B 0,C 180,E1 -13372.69,E2 -13372.69} C_VEL
LIN {X 0,Y 358.16,Z 615.045,A -85,B 0,C 180,E1 -13376.049,E2 -13376.049} C_VEL
LIN {X 0,Y 356.947,Z 625.831,A -85,B 0,C 180,E1 -13379.708,E2 -13379.708} C_VEL
LIN {X 0,Y 355.826,Z 637.71,A -85,B 0,C 180,E1 -13383.616,E2 -13383.616} C_VEL
LIN {X 0,Y 354.932,Z 649.324,A -85,B 0,C 180,E1 -13387.365,E2 -13387.365} C_VEL
LIN {X 0,Y 355.732,Z 656.694,A -85,B 0,C 180,E1 -13388.212,E2 -13388.212} C_VEL
LIN {X 0,Y 358.035,Z 667.079,A -85,B 0,C 180,E1 -13388.795,E2 -13388.795} C_VEL
LIN {X 0,Y 359.685,Z 679.466,A -85,B 0,C 180,E1 -13389.458,E2 -13389.458} C_VEL
LIN {X 0,Y 360.222,Z 692.334,A -85,B 0,C 180,E1 -13390.267,E2 -13390.267} C_VEL
LIN {X 0,Y 360.265,Z 704.629,A -85,B 0,C 180,E1 -13391.225,E2 -13391.225} C_VEL
LIN {X 0,Y 359.966,Z 711.007,A -85,B 0,C 180,E1 -13391.798,E2 -13391.798} C_VEL
LIN {X 0,Y 358.56,Z 723.234,A -85,B 0,C 180,E1 -13393.05,E2 -13393.05} C_VEL
LIN {X 0,Y 357.303,Z 733.089,A -85,B 0,C 180,E1 -13394.3,E2 -13394.3} C_VEL
LIN {X 0,Y 356.165,Z 742.24,A -85,B 0,C 180,E1 -13395.722,E2 -13395.722} C_VEL
LIN {X 0,Y 355.209,Z 751.205,A -85,B 0,C 180,E1 -13397.431,E2 -13397.431} C_VEL
LIN {X 0,Y 354.338,Z 758.514,A -85,B 0,C 180,E1 -13399.14,E2 -13399.14} C_VEL
LIN {X 0,Y 353.88,Z 764.397,A -85,B 0,C 180,E1 -13400.859,E2 -13400.859} C_VEL
LIN {X 0,Y 353.611,Z 769.055,A -85,B 0,C 180,E1 -13402.578,E2 -13402.578} C_VEL
LIN {X 0,Y 353.451,Z 772.603,A -85,B 0,C 180,E1 -13404.295,E2 -13404.295} C_VEL
LIN {X 0,Y 353.444,Z 774.39,A -85,B 0,C 180,E1 -13405.439,E2 -13405.439} C_VEL
LIN {X 0,Y 353.4,Z 775.758,A -85,B 0,C 180,E1 -13406.581,E2 -13406.581} C_VEL
LIN {X 0,Y 353.498,Z 776.679,A -85,B 0,C 180,E1 -13407.722,E2 -13407.722} C_VEL
LIN {X 0,Y 353.561,Z 777.16,A -85,B 0,C 180,E1 -13408.862,E2 -13408.862} C_VEL
LIN {X 0,Y 353.571,Z 777.228,A -85,B 0,C 180,E1 -13410.001,E2 -13410.001} C_VEL
LIN {X 0,Y 353.571,Z 776.875,A -85,B 0,C 180,E1 -13411.14,E2 -13411.14} C_VEL
LIN {X 0,Y 353.567,Z 776.049,A -85,B 0,C 180,E1 -13412.279,E2 -13412.279} C_VEL
LIN {X 0,Y 353.424,Z 774.789,A -85,B 0,C 180,E1 -13413.421,E2 -13413.421} C_VEL
LIN {X 0,Y 353.52,Z 772.069,A -85,B 0,C 180,E1 -13415.134,E2 -13415.134} C_VEL
LIN {X 0,Y 353.527,Z 768.245,A -85,B 0,C 180,E1 -13416.851,E2 -13416.851} C_VEL
LIN {X 0,Y 353.735,Z 763.238,A -85,B 0,C 180,E1 -13418.571,E2 -13418.571} C_VEL
LIN {X 0,Y 354.115,Z 756.887,A -85,B 0,C 180,E1 -13420.29,E2 -13420.29} C_VEL
LIN {X 0,Y 354.719,Z 748.889,A -85,B 0,C 180,E1 -13422.008,E2 -13422.008} C_VEL
LIN {X 0,Y 355.4,Z 740.731,A -85,B 0,C 180,E1 -13423.437,E2 -13423.437} C_VEL
LIN {X 0,Y 356.161,Z 731.422,A -85,B 0,C 180,E1 -13424.781,E2 -13424.781} C_VEL
LIN {X 0,Y 357.09,Z 721.049,A -85,B 0,C 180,E1 -13425.995,E2 -13425.995} C_VEL
LIN {X 0,Y 358.134,Z 708.916,A -85,B 0,C 180,E1 -13427.12,E2 -13427.12} C_VEL
LIN {X 0,Y 358.118,Z 702.368,A -85,B 0,C 180,E1 -13427.636,E2 -13427.636} C_VEL
LIN {X 0,Y 357.472,Z 688.925,A -85,B 0,C 180,E1 -13428.499,E2 -13428.499} C_VEL
LIN {X 0,Y 356.409,Z 675.341,A -85,B 0,C 180,E1 -13429.135,E2 -13429.135} C_VEL
LIN {X 0,Y 354.629,Z 658.047,A -85,B 0,C 180,E1 -13429.765,E2 -13429.765} C_VEL
LIN {X 0,Y 354.418,Z 654.642,A -85,B 0,C 180,E1 -13430.004,E2 -13430.004} C_VEL
LIN {X 0,Y 355.141,Z 640.011,A -85,B 0,C 180,E1 -13434.556,E2 -13434.556} C_VEL
LIN {X 0,Y 355.987,Z 628.236,A -85,B 0,C 180,E1 -13438.283,E2 -13438.283} C_VEL
LIN {X 0,Y 356.981,Z 616.115,A -85,B 0,C 180,E1 -13442.16,E2 -13442.16} C_VEL
LIN {X 0,Y 358.051,Z 605.259,A -85,B 0,C 180,E1 -13445.73,E2 -13445.73} C_VEL
LIN {X 0,Y 358.478,Z 600.187,A -85,B 0,C 180,E1 -13447.429,E2 -13447.429} C_VEL
LIN {X 0,Y 357.368,Z 593.294,A -85,B 0,C 180,E1 -13449.916,E2 -13449.916} C_VEL
LIN {X 0,Y 355.771,Z 585.084,A -85,B 0,C 180,E1 -13453.037,E2 -13453.037} C_VEL
LIN {X 0,Y 354.811,Z 580.291,A -85,B 0,C 180,E1 -13454.986,E2 -13454.986} C_VEL
LIN {X 0,Y 354.793,Z 580.293,A -85,B 0,C 180,E1 -13458.829,E2 -13458.829} C_VEL
LIN {X 0,Y 354.817,Z 580.289,A -85,B 0,C 180,E1 -13462.402,E2 -13462.402} C_VEL
LIN {X 0,Y 354.817,Z 580.285,A -85,B 0,C 180,E1 -13464.941,E2 -13464.941} C_VEL
LIN {X 0,Y 354.798,Z 580.292,A -85,B 0,C 180,E1 -13468.405,E2 -13468.405} C_VEL
LIN {X 0,Y 354.851,Z 580.281,A -85,B 0,C 180,E1 -13471.619,E2 -13471.619} C_VEL
LIN {X 0,Y 354.904,Z 580.278,A -85,B 0,C 180,E1 -13474.173,E2 -13474.173} C_VEL
LIN {X 0,Y 354.84,Z 580.284,A -85,B 0,C 180,E1 -13477.894,E2 -13477.894} C_VEL
LIN {X 0,Y 354.927,Z 580.273,A -85,B 0,C 180,E1 -13481.891,E2 -13481.891} C_VEL
LIN {X 0,Y 354.947,Z 580.271,A -85,B 0,C 180,E1 -13485.981,E2 -13485.981} C_VEL
LIN {X 0,Y 354.983,Z 580.265,A -85,B 0,C 180,E1 -13489.736,E2 -13489.736} C_VEL
LIN {X 0,Y 355.133,Z 580.248,A -85,B 0,C 180,E1 -13492.037,E2 -13492.037} C_VEL
LIN {X 0,Y 355.096,Z 580.255,A -85,B 0,C 180,E1 -13494.32,E2 -13494.32} C_VEL
LIN {X 0,Y 355.247,Z 580.232,A -85,B 0,C 180,E1 -13497.732,E2 -13497.732} C_VEL
LIN {X 0,Y 355.402,Z 580.214,A -85,B 0,C 180,E1 -13500,E2 -13500} C_VEL
LIN {X 0,Y 355.247,Z 580.236,A -85,B 0,C 180,E1 -13502.267,E2 -13502.267} C_VEL
LIN {X 0,Y 355.142,Z 580.246,A -85,B 0,C 180,E1 -13506.819,E2 -13506.819} C_VEL
LIN {X 0,Y 355.019,Z 580.26,A -85,B 0,C 180,E1 -13509.112,E2 -13509.112} C_VEL
LIN {X 0,Y 354.925,Z 580.275,A -85,B 0,C 180,E1 -13512.58,E2 -13512.58} C_VEL
LIN {X 0,Y 354.893,Z 580.278,A -85,B 0,C 180,E1 -13516.095,E2 -13516.095} C_VEL
LIN {X 0,Y 354.91,Z 580.279,A -85,B 0,C 180,E1 -13518.471,E2 -13518.471} C_VEL
LIN {X 0,Y 354.838,Z 580.285,A -85,B 0,C 180,E1 -13522.105,E2 -13522.105} C_VEL
LIN {X 0,Y 354.902,Z 580.275,A -85,B 0,C 180,E1 -13525.827,E2 -13525.827} C_VEL
LIN {X 0,Y 354.856,Z 580.28,A -85,B 0,C 180,E1 -13529.678,E2 -13529.678} C_VEL
LIN {X 0,Y 354.808,Z 580.286,A -85,B 0,C 180,E1 -13533.701,E2 -13533.701} C_VEL
LIN {X 0,Y 354.801,Z 580.292,A -85,B 0,C 180,E1 -13536.458,E2 -13536.458} C_VEL
LIN {X 0,Y 354.826,Z 580.283,A -85,B 0,C 180,E1 -13539.423,E2 -13539.423} C_VEL
LIN {X 0,Y 354.79,Z 580.29,A -85,B 0,C 180,E1 -13542.867,E2 -13542.867} C_VEL
LIN {X 0,Y 354.771,Z 580.292,A -85,B 0,C 180,E1 -13546.103,E2 -13546.103} C_VEL
LIN {X 0,Y 354.79,Z 580.288,A -85,B 0,C 180,E1 -13549.178,E2 -13549.178} C_VEL
LIN {X 0,Y 354.812,Z 580.29,A -85,B 0,C 180,E1 -13552.401,E2 -13552.401} C_VEL
LIN {X 0,Y 354.812,Z 580.287,A -85,B 0,C 180,E1 -13554.94,E2 -13554.94} C_VEL
LIN {X 0,Y 354.794,Z 580.292,A -85,B 0,C 180,E1 -13558.404,E2 -13558.404} C_VEL
LIN {X 0,Y 354.847,Z 580.281,A -85,B 0,C 180,E1 -13561.618,E2 -13561.618} C_VEL
LIN {X 0,Y 354.899,Z 580.277,A -85,B 0,C 180,E1 -13564.172,E2 -13564.172} C_VEL
LIN {X 0,Y 354.836,Z 580.283,A -85,B 0,C 180,E1 -13567.893,E2 -13567.893} C_VEL
LIN {X 0,Y 354.922,Z 580.272,A -85,B 0,C 180,E1 -13571.891,E2 -13571.891} C_VEL
LIN {X 0,Y 354.943,Z 580.27,A -85,B 0,C 180,E1 -13575.98,E2 -13575.98} C_VEL
LIN {X 0,Y 354.982,Z 580.264,A -85,B 0,C 180,E1 -13579.735,E2 -13579.735} C_VEL
LIN {X 0,Y 355.113,Z 580.249,A -85,B 0,C 180,E1 -13582.036,E2 -13582.036} C_VEL
LIN {X 0,Y 354.989,Z 580.266,A -85,B 0,C 180,E1 -13584.888,E2 -13584.888} C_VEL
LIN {X 0,Y 354.927,Z 580.273,A -85,B 0,C 180,E1 -13585.385,E2 -13585.385} C_VEL
LIN {X 0,Y 358.655,Z 592.367,A -85,B 0,C 180,E1 -13586.376,E2 -13586.376} C_VEL
LIN {X 0,Y 360.513,Z 600.104,A -85,B 0,C 180,E1 -13587.12,E2 -13587.12} C_VEL
LIN {X 0,Y 359.765,Z 610.823,A -85,B 0,C 180,E1 -13588.18,E2 -13588.18} C_VEL
LIN {X 0,Y 359.049,Z 620.354,A -85,B 0,C 180,E1 -13589.349,E2 -13589.349} C_VEL
LIN {X 0,Y 358.231,Z 629.857,A -85,B 0,C 180,E1 -13590.779,E2 -13590.779} C_VEL
LIN {X 0,Y 357.439,Z 637.812,A -85,B 0,C 180,E1 -13592.253,E2 -13592.253} C_VEL
LIN {X 0,Y 356.745,Z 645.233,A -85,B 0,C 180,E1 -13593.953,E2 -13593.953} C_VEL
LIN {X 0,Y 356.17,Z 651.212,A -85,B 0,C 180,E1 -13595.661,E2 -13595.661} C_VEL
LIN {X 0,Y 355.723,Z 655.957,A -85,B 0,C 180,E1 -13597.377,E2 -13597.377} C_VEL
LIN {X 0,Y 355.289,Z 659.625,A -85,B 0,C 180,E1 -13599.104,E2 -13599.104} C_VEL
LIN {X 0,Y 355.126,Z 661.516,A -85,B 0,C 180,E1 -13600.259,E2 -13600.259} C_VEL
LIN {X 0,Y 355.014,Z 662.938,A -85,B 0,C 180,E1 -13601.417,E2 -13601.417} C_VEL
LIN {X 0,Y 355.008,Z 664.589,A -85,B 0,C 180,E1 -13603.741,E2 -13603.741} C_VEL
LIN {X 0,Y 355.043,Z 664.809,A -85,B 0,C 180,E1 -13604.911,E2 -13604.911} C_VEL
LIN {X 0,Y 355.141,Z 664.6,A -85,B 0,C 180,E1 -13606.083,E2 -13606.083} C_VEL
LIN {X 0,Y 355.307,Z 663.997,A -85,B 0,C 180,E1 -13607.258,E2 -13607.258} C_VEL
LIN {X 0,Y 355.586,Z 662.984,A -85,B 0,C 180,E1 -13608.434,E2 -13608.434} C_VEL
LIN {X 0,Y 355.876,Z 661.498,A -85,B 0,C 180,E1 -13609.615,E2 -13609.615} C_VEL
LIN {X 0,Y 356.487,Z 658.43,A -85,B 0,C 180,E1 -13611.389,E2 -13611.389} C_VEL
LIN {X 0,Y 357.238,Z 654.225,A -85,B 0,C 180,E1 -13613.169,E2 -13613.169} C_VEL
LIN {X 0,Y 358.176,Z 648.74,A -85,B 0,C 180,E1 -13614.951,E2 -13614.951} C_VEL
LIN {X 0,Y 359.257,Z 641.767,A -85,B 0,C 180,E1 -13616.738,E2 -13616.738} C_VEL
LIN {X 0,Y 360.439,Z 633.828,A -85,B 0,C 180,E1 -13618.347,E2 -13618.347} C_VEL
LIN {X 0,Y 361.654,Z 624.555,A -85,B 0,C 180,E1 -13619.864,E2 -13619.864} C_VEL
LIN {X 0,Y 362.779,Z 614.366,A -85,B 0,C 180,E1 -13621.211,E2 -13621.211} C_VEL
LIN {X 0,Y 363.613,Z 605.535,A -85,B 0,C 180,E1 -13622.157,E2 -13622.157} C_VEL
LIN {X 0,Y 360.604,Z 595.739,A -85,B 0,C 180,E1 -13623.32,E2 -13623.32} C_VEL
LIN {X 0,Y 356.484,Z 584.672,A -85,B 0,C 180,E1 -13624.465,E2 -13624.465} C_VEL
LIN {X 0,Y 354.86,Z 580.284,A -85,B 0,C 180,E1 -13624.876,E2 -13624.876} C_VEL
LIN {X 0,Y 354.9,Z 580.376,A -85,B 0,C 180,E1 -13626.27,E2 -13626.27} C_VEL
LIN {X 0,Y 356.178,Z 587.888,A -85,B 0,C 180,E1 -13629.689,E2 -13629.689} C_VEL
LIN {X 0,Y 356.487,Z 592.159,A -85,B 0,C 180,E1 -13631.574,E2 -13631.574} C_VEL
LIN {X 0,Y 355.804,Z 594.311,A -85,B 0,C 180,E1 -13632.45,E2 -13632.45} C_VEL
LIN {X 0,Y 352.91,Z 598.098,A -85,B 0,C 180,E1 -13633.855,E2 -13633.855} C_VEL
LIN {X 0,Y 350.416,Z 601.15,A -85,B 0,C 180,E1 -13634.99,E2 -13634.99} C_VEL
LIN {X 0,Y 349.28,Z 603.366,A -85,B 0,C 180,E1 -13635.877,E2 -13635.877} C_VEL
LIN {X 0,Y 349.153,Z 604.075,A -85,B 0,C 180,E1 -13636.18,E2 -13636.18} C_VEL
LIN {X 0,Y 348.736,Z 612.824,A -85,B 0,C 180,E1 -13639.976,E2 -13639.976} C_VEL
LIN {X 0,Y 348.417,Z 620.615,A -85,B 0,C 180,E1 -13643.337,E2 -13643.337} C_VEL
LIN {X 0,Y 348.153,Z 627.758,A -85,B 0,C 180,E1 -13646.403,E2 -13646.403} C_VEL
LIN {X 0,Y 348.072,Z 629.628,A -85,B 0,C 180,E1 -13647.181,E2 -13647.181} C_VEL
LIN {X 0,Y 350.729,Z 642.956,A -85,B 0,C 180,E1 -13647.834,E2 -13647.834} C_VEL
LIN {X 0,Y 352.859,Z 654.838,A -85,B 0,C 180,E1 -13648.607,E2 -13648.607} C_VEL
LIN {X 0,Y 352.312,Z 666.227,A -85,B 0,C 180,E1 -13649.439,E2 -13649.439} C_VEL
LIN {X 0,Y 351.351,Z 677.68,A -85,B 0,C 180,E1 -13650.491,E2 -13650.491} C_VEL
LIN {X 0,Y 350.401,Z 688.407,A -85,B 0,C 180,E1 -13651.727,E2 -13651.727} C_VEL
LIN {X 0,Y 349.513,Z 698.147,A -85,B 0,C 180,E1 -13653.101,E2 -13653.101} C_VEL
LIN {X 0,Y 348.66,Z 707.053,A -85,B 0,C 180,E1 -13654.638,E2 -13654.638} C_VEL
LIN {X 0,Y 347.778,Z 715.654,A -85,B 0,C 180,E1 -13656.478,E2 -13656.478} C_VEL
LIN {X 0,Y 347.246,Z 722.508,A -85,B 0,C 180,E1 -13658.324,E2 -13658.324} C_VEL
LIN {X 0,Y 346.723,Z 728.6,A -85,B 0,C 180,E1 -13660.461,E2 -13660.461} C_VEL
LIN {X 0,Y 346.453,Z 732.751,A -85,B 0,C 180,E1 -13662.439,E2 -13662.439} C_VEL
LIN {X 0,Y 346.203,Z 735.852,A -85,B 0,C 180,E1 -13664.699,E2 -13664.699} C_VEL
LIN {X 0,Y 346.179,Z 736.883,A -85,B 0,C 180,E1 -13665.9,E2 -13665.9} C_VEL
LIN {X 0,Y 346.252,Z 737.433,A -85,B 0,C 180,E1 -13667.099,E2 -13667.099} C_VEL
LIN {X 0,Y 346.308,Z 737.555,A -85,B 0,C 180,E1 -13668.291,E2 -13668.291} C_VEL
LIN {X 0,Y 346.333,Z 737.278,A -85,B 0,C 180,E1 -13669.477,E2 -13669.477} C_VEL
LIN {X 0,Y 346.494,Z 736.548,A -85,B 0,C 180,E1 -13670.662,E2 -13670.662} C_VEL
LIN {X 0,Y 346.978,Z 733.905,A -85,B 0,C 180,E1 -13672.961,E2 -13672.961} C_VEL
LIN {X 0,Y 347.417,Z 730.642,A -85,B 0,C 180,E1 -13674.778,E2 -13674.778} C_VEL
LIN {X 0,Y 348.019,Z 726.402,A -85,B 0,C 180,E1 -13676.527,E2 -13676.527} C_VEL
LIN {X 0,Y 348.995,Z 719.917,A -85,B 0,C 180,E1 -13678.558,E2 -13678.558} C_VEL
LIN {X 0,Y 350.104,Z 712.881,A -85,B 0,C 180,E1 -13680.288,E2 -13680.288} C_VEL
LIN {X 0,Y 351.449,Z 704.203,A -85,B 0,C 180,E1 -13682.006,E2 -13682.006} C_VEL
LIN {X 0,Y 352.755,Z 695.352,A -85,B 0,C 180,E1 -13683.427,E2 -13683.427} C_VEL
LIN {X 0,Y 354.102,Z 685.719,A -85,B 0,C 180,E1 -13684.697,E2 -13684.697} C_VEL
LIN {X 0,Y 355.481,Z 674.051,A -85,B 0,C 180,E1 -13685.94,E2 -13685.94} C_VEL
LIN {X 0,Y 356.786,Z 662.096,A -85,B 0,C 180,E1 -13686.93,E2 -13686.93} C_VEL
LIN {X 0,Y 356.613,Z 658.605,A -85,B 0,C 180,E1 -13687.218,E2 -13687.218} C_VEL
LIN {X 0,Y 354.65,Z 648.369,A -85,B 0,C 180,E1 -13688.103,E2 -13688.103} C_VEL
LIN {X 0,Y 350.777,Z 636.095,A -85,B 0,C 180,E1 -13689.115,E2 -13689.115} C_VEL
LIN {X 0,Y 349.845,Z 633.298,A -85,B 0,C 180,E1 -13689.35,E2 -13689.35} C_VEL
LIN {X 0,Y 350.392,Z 625.711,A -85,B 0,C 180,E1 -13692.747,E2 -13692.747} C_VEL
LIN {X 0,Y 350.964,Z 617.908,A -85,B 0,C 180,E1 -13696.281,E2 -13696.281} C_VEL
LIN {X 0,Y 351.701,Z 609.648,A -85,B 0,C 180,E1 -13700.088,E2 -13700.088} C_VEL
LIN {X 0,Y 352.198,Z 604.885,A -85,B 0,C 180,E1 -13702.281,E2 -13702.281} C_VEL
LIN {X 0,Y 352.326,Z 600.943,A -85,B 0,C 180,E1 -13704.138,E2 -13704.138} C_VEL
LIN {X 0,Y 351.733,Z 596.178,A -85,B 0,C 180,E1 -13706.717,E2 -13706.717} C_VEL
LIN {X 0,Y 350.71,Z 591.439,A -85,B 0,C 180,E1 -13709.404,E2 -13709.404} C_VEL
LIN {X 0,Y 349.324,Z 586.144,A -85,B 0,C 180,E1 -13712.903,E2 -13712.903} C_VEL
LIN {X 0,Y 347.986,Z 582.232,A -85,B 0,C 180,E1 -13716.116,E2 -13716.116} C_VEL
LIN {X 0,Y 347.746,Z 581.168,A -85,B 0,C 180,E1 -13717.152,E2 -13717.152} C_VEL
LIN {X 0,Y 347.794,Z 581.164,A -85,B 0,C 180,E1 -13721.139,E2 -13721.139} C_VEL
LIN {X 0,Y 347.797,Z 581.2,A -85,B 0,C 180,E1 -13721.31,E2 -13721.31} C_VEL
LIN {X 0,Y 349.353,Z 588.313,A -85,B 0,C 180,E1 -13724.758,E2 -13724.758} C_VEL
LIN {X 0,Y 350.735,Z 595.234,A -85,B 0,C 180,E1 -13727.852,E2 -13727.852} C_VEL
LIN {X 0,Y 352.098,Z 602.169,A -85,B 0,C 180,E1 -13730.764,E2 -13730.764} C_VEL
LIN {X 0,Y 352.516,Z 606.438,A -85,B 0,C 180,E1 -13732.45,E2 -13732.45} C_VEL
LIN {X 0,Y 351.195,Z 616.114,A -85,B 0,C 180,E1 -13735.923,E2 -13735.923} C_VEL
LIN {X 0,Y 349.894,Z 627.116,A -85,B 0,C 180,E1 -13739.736,E2 -13739.736} C_VEL
LIN {X 0,Y 348.741,Z 638.804,A -85,B 0,C 180,E1 -13743.683,E2 -13743.683} C_VEL
LIN {X 0,Y 348.052,Z 647.223,A -85,B 0,C 180,E1 -13746.459,E2 -13746.459} C_VEL
LIN {X 0,Y 349.213,Z 656.649,A -85,B 0,C 180,E1 -13747.593,E2 -13747.593} C_VEL
LIN {X 0,Y 351.944,Z 669.28,A -85,B 0,C 180,E1 -13748.333,E2 -13748.333} C_VEL
LIN {X 0,Y 353.368,Z 681.661,A -85,B 0,C 180,E1 -13749.062,E2 -13749.062} C_VEL
LIN {X 0,Y 353.734,Z 694.351,A -85,B 0,C 180,E1 -13749.915,E2 -13749.915} C_VEL
LIN {X 0,Y 353.633,Z 707.337,A -85,B 0,C 180,E1 -13751.01,E2 -13751.01} C_VEL
LIN {X 0,Y 352.464,Z 718.848,A -85,B 0,C 180,E1 -13752.149,E2 -13752.149} C_VEL
LIN {X 0,Y 350.872,Z 730.385,A -85,B 0,C 180,E1 -13753.566,E2 -13753.566} C_VEL
LIN {X 0,Y 349.487,Z 740.767,A -85,B 0,C 180,E1 -13755.145,E2 -13755.145} C_VEL
LIN {X 0,Y 348.405,Z 749.896,A -85,B 0,C 180,E1 -13756.885,E2 -13756.885} C_VEL
LIN {X 0,Y 347.419,Z 757.349,A -85,B 0,C 180,E1 -13758.626,E2 -13758.626} C_VEL
LIN {X 0,Y 346.978,Z 762.433,A -85,B 0,C 180,E1 -13760.087,E2 -13760.087} C_VEL
LIN {X 0,Y 346.589,Z 767.417,A -85,B 0,C 180,E1 -13761.841,E2 -13761.841} C_VEL
LIN {X 0,Y 346.401,Z 771.672,A -85,B 0,C 180,E1 -13763.799,E2 -13763.799} C_VEL
LIN {X 0,Y 346.352,Z 774.08,A -85,B 0,C 180,E1 -13765.346,E2 -13765.346} C_VEL
LIN {X 0,Y 346.316,Z 775.419,A -85,B 0,C 180,E1 -13766.511,E2 -13766.511} C_VEL
LIN {X 0,Y 346.398,Z 776.29,A -85,B 0,C 180,E1 -13767.676,E2 -13767.676} C_VEL
LIN {X 0,Y 346.493,Z 776.748,A -85,B 0,C 180,E1 -13768.839,E2 -13768.839} C_VEL
LIN {X 0,Y 346.502,Z 776.792,A -85,B 0,C 180,E1 -13770.001,E2 -13770.001} C_VEL
LIN {X 0,Y 346.504,Z 776.393,A -85,B 0,C 180,E1 -13771.163,E2 -13771.163} C_VEL
LIN {X 0,Y 346.482,Z 775.538,A -85,B 0,C 180,E1 -13772.326,E2 -13772.326} C_VEL
LIN {X 0,Y 346.341,Z 774.254,A -85,B 0,C 180,E1 -13773.491,E2 -13773.491} C_VEL
LIN {X 0,Y 346.428,Z 771.484,A -85,B 0,C 180,E1 -13775.239,E2 -13775.239} C_VEL
LIN {X 0,Y 346.448,Z 767.607,A -85,B 0,C 180,E1 -13776.992,E2 -13776.992} C_VEL
LIN {X 0,Y 346.733,Z 761.544,A -85,B 0,C 180,E1 -13779.039,E2 -13779.039} C_VEL
LIN {X 0,Y 347.129,Z 754.837,A -85,B 0,C 180,E1 -13780.795,E2 -13780.795} C_VEL
LIN {X 0,Y 347.859,Z 746.501,A -85,B 0,C 180,E1 -13782.545,E2 -13782.545} C_VEL
LIN {X 0,Y 348.793,Z 736.581,A -85,B 0,C 180,E1 -13784.197,E2 -13784.197} C_VEL
LIN {X 0,Y 349.512,Z 727.353,A -85,B 0,C 180,E1 -13785.453,E2 -13785.453} C_VEL
LIN {X 0,Y 350.438,Z 716.982,A -85,B 0,C 180,E1 -13786.607,E2 -13786.607} C_VEL
LIN {X 0,Y 351.304,Z 705.561,A -85,B 0,C 180,E1 -13787.614,E2 -13787.614} C_VEL
LIN {X 0,Y 350.705,Z 692.539,A -85,B 0,C 180,E1 -13788.551,E2 -13788.551} C_VEL
LIN {X 0,Y 349.785,Z 679.108,A -85,B 0,C 180,E1 -13789.263,E2 -13789.263} C_VEL
LIN {X 0,Y 347.624,Z 657.367,A -85,B 0,C 180,E1 -13790.103,E2 -13790.103} C_VEL
LIN {X 0,Y 347.374,Z 653.411,A -85,B 0,C 180,E1 -13790.427,E2 -13790.427} C_VEL
LIN {X 0,Y 348.085,Z 640.04,A -85,B 0,C 180,E1 -13794.69,E2 -13794.69} C_VEL
LIN {X 0,Y 349.045,Z 627.038,A -85,B 0,C 180,E1 -13798.898,E2 -13798.898} C_VEL
LIN {X 0,Y 350.017,Z 616.058,A -85,B 0,C 180,E1 -13802.507,E2 -13802.507} C_VEL
LIN {X 0,Y 351.104,Z 605.111,A -85,B 0,C 180,E1 -13806.184,E2 -13806.184} C_VEL
LIN {X 0,Y 351.471,Z 601.048,A -85,B 0,C 180,E1 -13807.582,E2 -13807.582} C_VEL
LIN {X 0,Y 350.224,Z 593.703,A -85,B 0,C 180,E1 -13810.31,E2 -13810.31} C_VEL
LIN {X 0,Y 348.648,Z 585.565,A -85,B 0,C 180,E1 -13813.474,E2 -13813.474} C_VEL
LIN {X 0,Y 347.779,Z 581.165,A -85,B 0,C 180,E1 -13815.322,E2 -13815.322} C_VEL
LIN {X 0,Y 347.756,Z 581.169,A -85,B 0,C 180,E1 -13818.397,E2 -13818.397} C_VEL
LIN {X 0,Y 347.782,Z 581.164,A -85,B 0,C 180,E1 -13822.011,E2 -13822.011} C_VEL
LIN {X 0,Y 347.75,Z 581.165,A -85,B 0,C 180,E1 -13825.536,E2 -13825.536} C_VEL
LIN {X 0,Y 347.766,Z 581.163,A -85,B 0,C 180,E1 -13829.653,E2 -13829.653} C_VEL
LIN {X 0,Y 347.836,Z 581.154,A -85,B 0,C 180,E1 -13833.608,E2 -13833.608} C_VEL
LIN {X 0,Y 347.794,Z 581.164,A -85,B 0,C 180,E1 -13836.162,E2 -13836.162} C_VEL
LIN {X 0,Y 347.818,Z 581.158,A -85,B 0,C 180,E1 -13839.909,E2 -13839.909} C_VEL
LIN {X 0,Y 347.871,Z 581.156,A -85,B 0,C 180,E1 -13842.359,E2 -13842.359} C_VEL
LIN {X 0,Y 347.902,Z 581.148,A -85,B 0,C 180,E1 -13845.971,E2 -13845.971} C_VEL
LIN {X 0,Y 347.933,Z 581.142,A -85,B 0,C 180,E1 -13849.525,E2 -13849.525} C_VEL
LIN {X 0,Y 348.112,Z 581.12,A -85,B 0,C 180,E1 -13853.042,E2 -13853.042} C_VEL
LIN {X 0,Y 348.21,Z 581.108,A -85,B 0,C 180,E1 -13857.686,E2 -13857.686} C_VEL
LIN {X 0,Y 348.35,Z 581.092,A -85,B 0,C 180,E1 -13860,E2 -13860} C_VEL
LIN {X 0,Y 348.21,Z 581.113,A -85,B 0,C 180,E1 -13862.313,E2 -13862.313} C_VEL
LIN {X 0,Y 348.11,Z 581.121,A -85,B 0,C 180,E1 -13866.957,E2 -13866.957} C_VEL
LIN {X 0,Y 347.971,Z 581.137,A -85,B 0,C 180,E1 -13869.298,E2 -13869.298} C_VEL
LIN {X 0,Y 347.894,Z 581.149,A -85,B 0,C 180,E1 -13872.839,E2 -13872.839} C_VEL
LIN {X 0,Y 347.843,Z 581.159,A -85,B 0,C 180,E1 -13876.431,E2 -13876.431} C_VEL
LIN {X 0,Y 347.859,Z 581.153,A -85,B 0,C 180,E1 -13878.86,E2 -13878.86} C_VEL
LIN {X 0,Y 347.777,Z 581.166,A -85,B 0,C 180,E1 -13882.579,E2 -13882.579} C_VEL
LIN {X 0,Y 347.815,Z 581.157,A -85,B 0,C 180,E1 -13885.108,E2 -13885.108} C_VEL
LIN {X 0,Y 347.813,Z 581.157,A -85,B 0,C 180,E1 -13887.693,E2 -13887.693} C_VEL
LIN {X 0,Y 347.766,Z 581.168,A -85,B 0,C 180,E1 -13890.346,E2 -13890.346} C_VEL
LIN {X 0,Y 347.746,Z 581.171,A -85,B 0,C 180,E1 -13894.463,E2 -13894.463} C_VEL
LIN {X 0,Y 347.776,Z 581.163,A -85,B 0,C 180,E1 -13897.988,E2 -13897.988} C_VEL
LIN {X 0,Y 347.752,Z 581.165,A -85,B 0,C 180,E1 -13901.829,E2 -13901.829} C_VEL
LIN {X 0,Y 347.767,Z 581.164,A -85,B 0,C 180,E1 -13905.016,E2 -13905.016} C_VEL
LIN {X 0,Y 347.752,Z 581.169,A -85,B 0,C 180,E1 -13908.396,E2 -13908.396} C_VEL
LIN {X 0,Y 347.777,Z 581.163,A -85,B 0,C 180,E1 -13912.01,E2 -13912.01} C_VEL
LIN {X 0,Y 347.745,Z 581.165,A -85,B 0,C 180,E1 -13915.535,E2 -13915.535} C_VEL
LIN {X 0,Y 347.745,Z 581.169,A -85,B 0,C 180,E1 -13918.3,E2 -13918.3} C_VEL
LIN {X 0,Y 347.779,Z 581.163,A -85,B 0,C 180,E1 -13920.987,E2 -13920.987} C_VEL
LIN {X 0,Y 347.831,Z 581.154,A -85,B 0,C 180,E1 -13923.607,E2 -13923.607} C_VEL
LIN {X 0,Y 347.789,Z 581.162,A -85,B 0,C 180,E1 -13926.161,E2 -13926.161} C_VEL
LIN {X 0,Y 347.813,Z 581.157,A -85,B 0,C 180,E1 -13929.908,E2 -13929.908} C_VEL
LIN {X 0,Y 347.866,Z 581.154,A -85,B 0,C 180,E1 -13932.358,E2 -13932.358} C_VEL
LIN {X 0,Y 347.897,Z 581.147,A -85,B 0,C 180,E1 -13935.97,E2 -13935.97} C_VEL
LIN {X 0,Y 347.932,Z 581.142,A -85,B 0,C 180,E1 -13939.525,E2 -13939.525} C_VEL
LIN {X 0,Y 348.074,Z 581.125,A -85,B 0,C 180,E1 -13941.874,E2 -13941.874} C_VEL
LIN {X 0,Y 347.959,Z 581.143,A -85,B 0,C 180,E1 -13944.784,E2 -13944.784} C_VEL
LIN {X 0,Y 347.949,Z 581.261,A -85,B 0,C 180,E1 -13945.074,E2 -13945.074} C_VEL
LIN {X 0,Y 351.338,Z 592.261,A -85,B 0,C 180,E1 -13945.985,E2 -13945.985} C_VEL
LIN {X 0,Y 353.64,Z 600.785,A -85,B 0,C 180,E1 -13946.822,E2 -13946.822} C_VEL
LIN {X 0,Y 352.854,Z 612.42,A -85,B 0,C 180,E1 -13948.001,E2 -13948.001} C_VEL
LIN {X 0,Y 352.04,Z 623.051,A -85,B 0,C 180,E1 -13949.363,E2 -13949.363} C_VEL
LIN {X 0,Y 351.076,Z 633.011,A -85,B 0,C 180,E1 -13950.966,E2 -13950.966} C_VEL
LIN {X 0,Y 350.299,Z 641.127,A -85,B 0,C 180,E1 -13952.586,E2 -13952.586} C_VEL
LIN {X 0,Y 349.587,Z 648.126,A -85,B 0,C 180,E1 -13954.322,E2 -13954.322} C_VEL
LIN {X 0,Y 348.913,Z 654.53,A -85,B 0,C 180,E1 -13956.359,E2 -13956.359} C_VEL
LIN {X 0,Y 348.48,Z 658.767,A -85,B 0,C 180,E1 -13958.115,E2 -13958.115} C_VEL
LIN {X 0,Y 348.23,Z 661.032,A -85,B 0,C 180,E1 -13959.29,E2 -13959.29} C_VEL
LIN {X 0,Y 348.077,Z 662.807,A -85,B 0,C 180,E1 -13960.469,E2 -13960.469} C_VEL
LIN {X 0,Y 347.938,Z 665.13,A -85,B 0,C 180,E1 -13962.836,E2 -13962.836} C_VEL
LIN {X 0,Y 347.974,Z 665.715,A -85,B 0,C 180,E1 -13964.2,E2 -13964.2} C_VEL
LIN {X 0,Y 348.168,Z 665.541,A -85,B 0,C 180,E1 -13966.414,E2 -13966.414} C_VEL
LIN {X 0,Y 348.634,Z 663.934,A -85,B 0,C 180,E1 -13968.657,E2 -13968.657} C_VEL
LIN {X 0,Y 349.007,Z 662.197,A -85,B 0,C 180,E1 -13970.018,E2 -13970.018} C_VEL
LIN {X 0,Y 349.701,Z 658.997,A -85,B 0,C 180,E1 -13971.825,E2 -13971.825} C_VEL
LIN {X 0,Y 350.5,Z 654.655,A -85,B 0,C 180,E1 -13973.641,E2 -13973.641} C_VEL
LIN {X 0,Y 351.458,Z 649.192,A -85,B 0,C 180,E1 -13975.408,E2 -13975.408} C_VEL
LIN {X 0,Y 352.466,Z 643.137,A -85,B 0,C 180,E1 -13976.975,E2 -13976.975} C_VEL
LIN {X 0,Y 353.587,Z 635.977,A -85,B 0,C 180,E1 -13978.49,E2 -13978.49} C_VEL
LIN {X 0,Y 354.866,Z 627.153,A -85,B 0,C 180,E1 -13980.003,E2 -13980.003} C_VEL
LIN {X 0,Y 355.978,Z 617.557,A -85,B 0,C 180,E1 -13981.344,E2 -13981.344} C_VEL
LIN {X 0,Y 356.991,Z 608.554,A -85,B 0,C 180,E1 -13982.365,E2 -13982.365} C_VEL
LIN {X 0,Y 356.405,Z 605.171,A -85,B 0,C 180,E1 -13982.78,E2 -13982.78} C_VEL
LIN {X 0,Y 353.123,Z 595.116,A -85,B 0,C 180,E1 -13983.985,E2 -13983.985} C_VEL
LIN {X 0,Y 349.273,Z 584.986,A -85,B 0,C 180,E1 -13985.05,E2 -13985.05} C_VEL
LIN {X 0,Y 347.803,Z 581.162,A -85,B 0,C 180,E1 -13985.455,E2 -13985.455} C_VEL
LIN {X 0,Y 347.852,Z 581.223,A -85,B 0,C 180,E1 -13985.977,E2 -13985.977} C_VEL
LIN {X 0,Y 349.106,Z 588.589,A -85,B 0,C 180,E1 -13989.354,E2 -13989.354} C_VEL
LIN {X 0,Y 349.527,Z 593.504,A -85,B 0,C 180,E1 -13991.568,E2 -13991.568} C_VEL
LIN {X 0,Y 349.241,Z 601.891,A -85,B 0,C 180,E1 -13995.226,E2 -13995.226} C_VEL
LIN {X 0,Y 349.153,Z 604.075,A -85,B 0,C 180,E1 -13996.18,E2 -13996.18} C_VEL
LIN {X 0,Y 348.366,Z 606.256,A -85,B 0,C 180,E1 -13997.073,E2 -13997.073} C_VEL
LIN {X 0,Y 342.374,Z 613.87,A -85,B 0,C 180,E1 -13999.952,E2 -13999.952} C_VEL
LIN {X 0,Y 341.646,Z 616.061,A -85,B 0,C 180,E1 -14000.869,E2 -14000.869} C_VEL
LIN {X 0,Y 341.335,Z 623.485,A -85,B 0,C 180,E1 -14004.1,E2 -14004.1} C_VEL
LIN {X 0,Y 341.081,Z 629.887,A -85,B 0,C 180,E1 -14006.873,E2 -14006.873} C_VEL
LIN {X 0,Y 343.68,Z 643.312,A -85,B 0,C 180,E1 -14007.546,E2 -14007.546} C_VEL
LIN {X 0,Y 345.89,Z 655.564,A -85,B 0,C 180,E1 -14008.368,E2 -14008.368} C_VEL
LIN {X 0,Y 345.294,Z 667.666,A -85,B 0,C 180,E1 -14009.284,E2 -14009.284} C_VEL
LIN {X 0,Y 344.209,Z 680.09,A -85,B 0,C 180,E1 -14010.49,E2 -14010.49} C_VEL
LIN {X 0,Y 343.353,Z 689.756,A -85,B 0,C 180,E1 -14011.658,E2 -14011.658} C_VEL
LIN {X 0,Y 342.346,Z 699.89,A -85,B 0,C 180,E1 -14013.152,E2 -14013.152} C_VEL
LIN {X 0,Y 341.4,Z 709.567,A -85,B 0,C 180,E1 -14014.924,E2 -14014.924} C_VEL
LIN {X 0,Y 340.665,Z 716.975,A -85,B 0,C 180,E1 -14016.602,E2 -14016.602} C_VEL
LIN {X 0,Y 340.129,Z 723.356,A -85,B 0,C 180,E1 -14018.403,E2 -14018.403} C_VEL
LIN {X 0,Y 339.733,Z 728.031,A -85,B 0,C 180,E1 -14020.042,E2 -14020.042} C_VEL
LIN {X 0,Y 339.397,Z 732.833,A -85,B 0,C 180,E1 -14022.271,E2 -14022.271} C_VEL
LIN {X 0,Y 339.128,Z 735.879,A -85,B 0,C 180,E1 -14024.371,E2 -14024.371} C_VEL
LIN {X 0,Y 339.102,Z 737.02,A -85,B 0,C 180,E1 -14025.6,E2 -14025.6} C_VEL
LIN {X 0,Y 339.163,Z 737.767,A -85,B 0,C 180,E1 -14026.877,E2 -14026.877} C_VEL
LIN {X 0,Y 339.201,Z 738.015,A -85,B 0,C 180,E1 -14028.043,E2 -14028.043} C_VEL
LIN {X 0,Y 339.236,Z 737.845,A -85,B 0,C 180,E1 -14029.255,E2 -14029.255} C_VEL
LIN {X 0,Y 339.403,Z 737.271,A -85,B 0,C 180,E1 -14030.465,E2 -14030.465} C_VEL
LIN {X 0,Y 339.623,Z 736.28,A -85,B 0,C 180,E1 -14031.672,E2 -14031.672} C_VEL
LIN {X 0,Y 339.91,Z 734.731,A -85,B 0,C 180,E1 -14032.942,E2 -14032.942} C_VEL
LIN {X 0,Y 340.32,Z 731.871,A -85,B 0,C 180,E1 -14034.668,E2 -14034.668} C_VEL
LIN {X 0,Y 340.923,Z 727.865,A -85,B 0,C 180,E1 -14036.455,E2 -14036.455} C_VEL
LIN {X 0,Y 341.811,Z 722.692,A -85,B 0,C 180,E1 -14038.233,E2 -14038.233} C_VEL
LIN {X 0,Y 342.878,Z 716.279,A -85,B 0,C 180,E1 -14040,E2 -14040} C_VEL
LIN {X 0,Y 344.296,Z 707.996,A -85,B 0,C 180,E1 -14041.814,E2 -14041.814} C_VEL
LIN {X 0,Y 345.836,Z 698.399,A -85,B 0,C 180,E1 -14043.496,E2 -14043.496} C_VEL
LIN {X 0,Y 347.322,Z 688.178,A -85,B 0,C 180,E1 -14044.934,E2 -14044.934} C_VEL
LIN {X 0,Y 348.868,Z 676.873,A -85,B 0,C 180,E1 -14046.217,E2 -14046.217} C_VEL
LIN {X 0,Y 350.216,Z 665.356,A -85,B 0,C 180,E1 -14047.254,E2 -14047.254} C_VEL
LIN {X 0,Y 350.45,Z 661.277,A -85,B 0,C 180,E1 -14047.586,E2 -14047.586} C_VEL
LIN {X 0,Y 348.293,Z 649.998,A -85,B 0,C 180,E1 -14048.616,E2 -14048.616} C_VEL
LIN {X 0,Y 344.244,Z 636.945,A -85,B 0,C 180,E1 -14049.765,E2 -14049.765} C_VEL
LIN {X 0,Y 343.131,Z 633.848,A -85,B 0,C 180,E1 -14050.038,E2 -14050.038} C_VEL
LIN {X 0,Y 343.725,Z 626.101,A -85,B 0,C 180,E1 -14053.6,E2 -14053.6} C_VEL
LIN {X 0,Y 344.393,Z 618.297,A -85,B 0,C 180,E1 -14057.212,E2 -14057.212} C_VEL
LIN {X 0,Y 345.188,Z 610.485,A -85,B 0,C 180,E1 -14060.873,E2 -14060.873} C_VEL
LIN {X 0,Y 345.732,Z 605.022,A -85,B 0,C 180,E1 -14063.512,E2 -14063.512} C_VEL
LIN {X 0,Y 345.603,Z 601.661,A -85,B 0,C 180,E1 -14065.281,E2 -14065.281} C_VEL
LIN {X 0,Y 345.079,Z 598.145,A -85,B 0,C 180,E1 -14067.274,E2 -14067.274} C_VEL
LIN {X 0,Y 344.143,Z 593.666,A -85,B 0,C 180,E1 -14070.023,E2 -14070.023} C_VEL
LIN {X 0,Y 342.861,Z 588.784,A -85,B 0,C 180,E1 -14073.604,E2 -14073.604} C_VEL
LIN {X 0,Y 341.793,Z 585.408,A -85,B 0,C 180,E1 -14076.688,E2 -14076.688} C_VEL
LIN {X 0,Y 340.835,Z 582.377,A -85,B 0,C 180,E1 -14080.823,E2 -14080.823} C_VEL
LIN {X 0,Y 342.326,Z 589.264,A -85,B 0,C 180,E1 -14084.269,E2 -14084.269} C_VEL
LIN {X 0,Y 343.757,Z 596.42,A -85,B 0,C 180,E1 -14087.573,E2 -14087.573} C_VEL
LIN {X 0,Y 345.256,Z 604.109,A -85,B 0,C 180,E1 -14090.875,E2 -14090.875} C_VEL
LIN {X 0,Y 345.548,Z 608.164,A -85,B 0,C 180,E1 -14092.487,E2 -14092.487} C_VEL
LIN {X 0,Y 344.213,Z 617.318,A -85,B 0,C 180,E1 -14095.843,E2 -14095.843} C_VEL
LIN {X 0,Y 342.952,Z 627.295,A -85,B 0,C 180,E1 -14099.395,E2 -14099.395} C_VEL
LIN {X 0,Y 341.828,Z 638.039,A -85,B 0,C 180,E1 -14103.109,E2 -14103.109} C_VEL
LIN {X 0,Y 341.269,Z 644.884,A -85,B 0,C 180,E1 -14105.404,E2 -14105.404} C_VEL
LIN {X 0,Y 342.567,Z 656.379,A -85,B 0,C 180,E1 -14106.901,E2 -14106.901} C_VEL
LIN {X 0,Y 345.728,Z 670.742,A -85,B 0,C 180,E1 -14107.812,E2 -14107.812} C_VEL
LIN {X 0,Y 347.048,Z 682.627,A -85,B 0,C 180,E1 -14108.557,E2 -14108.557} C_VEL
LIN {X 0,Y 347.252,Z 695.161,A -85,B 0,C 180,E1 -14109.457,E2 -14109.457} C_VEL
LIN {X 0,Y 347.013,Z 708.414,A -85,B 0,C 180,E1 -14110.633,E2 -14110.633} C_VEL
LIN {X 0,Y 345.579,Z 720.794,A -85,B 0,C 180,E1 -14111.934,E2 -14111.934} C_VEL
LIN {X 0,Y 343.959,Z 731.925,A -85,B 0,C 180,E1 -14113.379,E2 -14113.379} C_VEL
LIN {X 0,Y 342.621,Z 741.085,A -85,B 0,C 180,E1 -14114.856,E2 -14114.856} C_VEL
LIN {X 0,Y 341.464,Z 749.969,A -85,B 0,C 180,E1 -14116.613,E2 -14116.613} C_VEL
LIN {X 0,Y 340.438,Z 757.332,A -85,B 0,C 180,E1 -14118.389,E2 -14118.389} C_VEL
LIN {X 0,Y 339.792,Z 764.1,A -85,B 0,C 180,E1 -14120.477,E2 -14120.477} C_VEL
LIN {X 0,Y 339.443,Z 768.614,A -85,B 0,C 180,E1 -14122.267,E2 -14122.267} C_VEL
LIN {X 0,Y 339.279,Z 772.039,A -85,B 0,C 180,E1 -14124.056,E2 -14124.056} C_VEL
LIN {X 0,Y 339.263,Z 773.773,A -85,B 0,C 180,E1 -14125.248,E2 -14125.248} C_VEL
LIN {X 0,Y 339.234,Z 775.064,A -85,B 0,C 180,E1 -14126.438,E2 -14126.438} C_VEL
LIN {X 0,Y 339.298,Z 775.903,A -85,B 0,C 180,E1 -14127.627,E2 -14127.627} C_VEL
LIN {X 0,Y 339.425,Z 776.338,A -85,B 0,C 180,E1 -14128.815,E2 -14128.815} C_VEL
LIN {X 0,Y 339.435,Z 776.352,A -85,B 0,C 180,E1 -14130.001,E2 -14130.001} C_VEL
LIN {X 0,Y 339.439,Z 775.896,A -85,B 0,C 180,E1 -14131.187,E2 -14131.187} C_VEL
LIN {X 0,Y 339.384,Z 775.008,A -85,B 0,C 180,E1 -14132.375,E2 -14132.375} C_VEL
LIN {X 0,Y 339.262,Z 773.696,A -85,B 0,C 180,E1 -14133.564,E2 -14133.564} C_VEL
LIN {X 0,Y 339.341,Z 770.858,A -85,B 0,C 180,E1 -14135.349,E2 -14135.349} C_VEL
LIN {X 0,Y 339.394,Z 766.911,A -85,B 0,C 180,E1 -14137.138,E2 -14137.138} C_VEL
LIN {X 0,Y 339.681,Z 760.736,A -85,B 0,C 180,E1 -14139.228,E2 -14139.228} C_VEL
LIN {X 0,Y 340.089,Z 753.945,A -85,B 0,C 180,E1 -14141.021,E2 -14141.021} C_VEL
LIN {X 0,Y 340.725,Z 747.017,A -85,B 0,C 180,E1 -14142.509,E2 -14142.509} C_VEL
LIN {X 0,Y 341.555,Z 738.675,A -85,B 0,C 180,E1 -14143.992,E2 -14143.992} C_VEL
LIN {X 0,Y 342.216,Z 729.965,A -85,B 0,C 180,E1 -14145.274,E2 -14145.274} C_VEL
LIN {X 0,Y 343.335,Z 718.329,A -85,B 0,C 180,E1 -14146.654,E2 -14146.654} C_VEL
LIN {X 0,Y 344.284,Z 707.503,A -85,B 0,C 180,E1 -14147.678,E2 -14147.678} C_VEL
LIN {X 0,Y 343.847,Z 695.188,A -85,B 0,C 180,E1 -14148.625,E2 -14148.625} C_VEL
LIN {X 0,Y 343.036,Z 681.485,A -85,B 0,C 180,E1 -14149.425,E2 -14149.425} C_VEL
LIN {X 0,Y 341.526,Z 665.082,A -85,B 0,C 180,E1 -14150.085,E2 -14150.085} C_VEL
LIN {X 0,Y 340.708,Z 657.963,A -85,B 0,C 180,E1 -14150.371,E2 -14150.371} C_VEL
LIN {X 0,Y 340.344,Z 652.278,A -85,B 0,C 180,E1 -14150.829,E2 -14150.829} C_VEL
LIN {X 0,Y 341.081,Z 638.817,A -85,B 0,C 180,E1 -14155.231,E2 -14155.231} C_VEL
LIN {X 0,Y 341.956,Z 627.81,A -85,B 0,C 180,E1 -14158.881,E2 -14158.881} C_VEL
LIN {X 0,Y 342.859,Z 617.902,A -85,B 0,C 180,E1 -14162.206,E2 -14162.206} C_VEL
LIN {X 0,Y 343.947,Z 607.783,A -85,B 0,C 180,E1 -14165.67,E2 -14165.67} C_VEL
LIN {X 0,Y 344.458,Z 601.907,A -85,B 0,C 180,E1 -14167.742,E2 -14167.742} C_VEL
LIN {X 0,Y 342.95,Z 593.403,A -85,B 0,C 180,E1 -14170.979,E2 -14170.979} C_VEL
LIN {X 0,Y 341.246,Z 584.799,A -85,B 0,C 180,E1 -14174.447,E2 -14174.447} C_VEL
LIN {X 0,Y 340.706,Z 582.045,A -85,B 0,C 180,E1 -14175.68,E2 -14175.68} C_VEL
LIN {X 0,Y 340.691,Z 582.049,A -85,B 0,C 180,E1 -14178.691,E2 -14178.691} C_VEL
LIN {X 0,Y 340.741,Z 582.039,A -85,B 0,C 180,E1 -14181.773,E2 -14181.773} C_VEL
LIN {X 0,Y 340.728,Z 582.039,A -85,B 0,C 180,E1 -14185.595,E2 -14185.595} C_VEL
LIN {X 0,Y 340.774,Z 582.036,A -85,B 0,C 180,E1 -14190.021,E2 -14190.021} C_VEL
LIN {X 0,Y 340.808,Z 582.029,A -85,B 0,C 180,E1 -14193.02,E2 -14193.02} C_VEL
LIN {X 0,Y 340.761,Z 582.035,A -85,B 0,C 180,E1 -14195.638,E2 -14195.638} C_VEL
LIN {X 0,Y 340.75,Z 582.036,A -85,B 0,C 180,E1 -14199.474,E2 -14199.474} C_VEL
LIN {X 0,Y 340.863,Z 582.025,A -85,B 0,C 180,E1 -14201.984,E2 -14201.984} C_VEL
LIN {X 0,Y 340.874,Z 582.021,A -85,B 0,C 180,E1 -14205.705,E2 -14205.705} C_VEL
LIN {X 0,Y 340.876,Z 582.021,A -85,B 0,C 180,E1 -14209.306,E2 -14209.306} C_VEL
LIN {X 0,Y 341.082,Z 581.996,A -85,B 0,C 180,E1 -14212.898,E2 -14212.898} C_VEL
LIN {X 0,Y 341.172,Z 581.984,A -85,B 0,C 180,E1 -14217.638,E2 -14217.638} C_VEL
LIN {X 0,Y 341.301,Z 581.97,A -85,B 0,C 180,E1 -14220,E2 -14220} C_VEL
LIN {X 0,Y 341.171,Z 581.99,A -85,B 0,C 180,E1 -14222.361,E2 -14222.361} C_VEL
LIN {X 0,Y 341.079,Z 581.996,A -85,B 0,C 180,E1 -14227.101,E2 -14227.101} C_VEL
LIN {X 0,Y 340.874,Z 582.024,A -85,B 0,C 180,E1 -14230.693,E2 -14230.693} C_VEL
LIN {X 0,Y 340.867,Z 582.027,A -85,B 0,C 180,E1 -14234.324,E2 -14234.324} C_VEL
LIN {X 0,Y 340.841,Z 582.031,A -85,B 0,C 180,E1 -14238.466,E2 -14238.466} C_VEL
LIN {X 0,Y 340.757,Z 582.036,A -85,B 0,C 180,E1 -14241.856,E2 -14241.856} C_VEL
LIN {X 0,Y 340.776,Z 582.033,A -85,B 0,C 180,E1 -14245.664,E2 -14245.664} C_VEL
LIN {X 0,Y 340.744,Z 582.042,A -85,B 0,C 180,E1 -14248.319,E2 -14248.319} C_VEL
LIN {X 0,Y 340.706,Z 582.043,A -85,B 0,C 180,E1 -14251.043,E2 -14251.043} C_VEL
LIN {X 0,Y 340.72,Z 582.04,A -85,B 0,C 180,E1 -14255.278,E2 -14255.278} C_VEL
LIN {X 0,Y 340.712,Z 582.046,A -85,B 0,C 180,E1 -14258.385,E2 -14258.385} C_VEL
LIN {X 0,Y 340.701,Z 582.044,A -85,B 0,C 180,E1 -14262.045,E2 -14262.045} C_VEL
LIN {X 0,Y 340.684,Z 582.044,A -85,B 0,C 180,E1 -14265.46,E2 -14265.46} C_VEL
LIN {X 0,Y 340.687,Z 582.048,A -85,B 0,C 180,E1 -14268.69,E2 -14268.69} C_VEL
LIN {X 0,Y 340.736,Z 582.038,A -85,B 0,C 180,E1 -14271.772,E2 -14271.772} C_VEL
LIN {X 0,Y 340.723,Z 582.039,A -85,B 0,C 180,E1 -14275.594,E2 -14275.594} C_VEL
LIN {X 0,Y 340.698,Z 582.045,A -85,B 0,C 180,E1 -14278.954,E2 -14278.954} C_VEL
LIN {X 0,Y 340.803,Z 582.031,A -85,B 0,C 180,E1 -14283.019,E2 -14283.019} C_VEL
LIN {X 0,Y 340.73,Z 582.041,A -85,B 0,C 180,E1 -14286.926,E2 -14286.926} C_VEL
LIN {X 0,Y 340.791,Z 582.036,A -85,B 0,C 180,E1 -14290.733,E2 -14290.733} C_VEL
LIN {X 0,Y 340.786,Z 582.032,A -85,B 0,C 180,E1 -14293.218,E2 -14293.218} C_VEL
LIN {X 0,Y 340.846,Z 582.027,A -85,B 0,C 180,E1 -14296.89,E2 -14296.89} C_VEL
LIN {X 0,Y 340.929,Z 582.019,A -85,B 0,C 180,E1 -14300.507,E2 -14300.507} C_VEL
LIN {X 0,Y 341.075,Z 581.999,A -85,B 0,C 180,E1 -14302.897,E2 -14302.897} C_VEL
LIN {X 0,Y 340.923,Z 582.02,A -85,B 0,C 180,E1 -14304.713,E2 -14304.713} C_VEL
LIN {X 0,Y 344.668,Z 594.379,A -85,B 0,C 180,E1 -14305.79,E2 -14305.79} C_VEL
LIN {X 0,Y 346.811,Z 602.342,A -85,B 0,C 180,E1 -14306.603,E2 -14306.603} C_VEL
LIN {X 0,Y 345.965,Z 613.984,A -85,B 0,C 180,E1 -14307.816,E2 -14307.816} C_VEL
LIN {X 0,Y 345.172,Z 623.822,A -85,B 0,C 180,E1 -14309.105,E2 -14309.105} C_VEL
LIN {X 0,Y 344.309,Z 632.649,A -85,B 0,C 180,E1 -14310.525,E2 -14310.525} C_VEL
LIN {X 0,Y 343.381,Z 641.767,A -85,B 0,C 180,E1 -14312.345,E2 -14312.345} C_VEL
LIN {X 0,Y 342.644,Z 648.853,A -85,B 0,C 180,E1 -14314.116,E2 -14314.116} C_VEL
LIN {X 0,Y 342.029,Z 654.512,A -85,B 0,C 180,E1 -14315.896,E2 -14315.896} C_VEL
LIN {X 0,Y 341.558,Z 658.98,A -85,B 0,C 180,E1 -14317.685,E2 -14317.685} C_VEL
LIN {X 0,Y 341.179,Z 662.391,A -85,B 0,C 180,E1 -14319.484,E2 -14319.484} C_VEL
LIN {X 0,Y 341.03,Z 664.091,A -85,B 0,C 180,E1 -14320.688,E2 -14320.688} C_VEL
LIN {X 0,Y 340.949,Z 665.39,A -85,B 0,C 180,E1 -14321.894,E2 -14321.894} C_VEL
LIN {X 0,Y 340.915,Z 666.287,A -85,B 0,C 180,E1 -14323.106,E2 -14323.106} C_VEL
LIN {X 0,Y 341.067,Z 666.804,A -85,B 0,C 180,E1 -14325.537,E2 -14325.537} C_VEL
LIN {X 0,Y 341.196,Z 666.484,A -85,B 0,C 180,E1 -14326.759,E2 -14326.759} C_VEL
LIN {X 0,Y 341.697,Z 664.875,A -85,B 0,C 180,E1 -14328.895,E2 -14328.895} C_VEL
LIN {X 0,Y 342.384,Z 661.902,A -85,B 0,C 180,E1 -14331.051,E2 -14331.051} C_VEL
LIN {X 0,Y 343.168,Z 658.202,A -85,B 0,C 180,E1 -14332.898,E2 -14332.898} C_VEL
LIN {X 0,Y 344.103,Z 653.294,A -85,B 0,C 180,E1 -14334.751,E2 -14334.751} C_VEL
LIN {X 0,Y 345.234,Z 647.004,A -85,B 0,C 180,E1 -14336.605,E2 -14336.605} C_VEL
LIN {X 0,Y 346.6,Z 638.955,A -85,B 0,C 180,E1 -14338.456,E2 -14338.456} C_VEL
LIN {X 0,Y 347.976,Z 630.251,A -85,B 0,C 180,E1 -14340.056,E2 -14340.056} C_VEL
LIN {X 0,Y 349.224,Z 620.237,A -85,B 0,C 180,E1 -14341.548,E2 -14341.548} C_VEL
LIN {X 0,Y 350.429,Z 609.736,A -85,B 0,C 180,E1 -14342.784,E2 -14342.784} C_VEL
LIN {X 0,Y 347.634,Z 600.132,A -85,B 0,C 180,E1 -14344.017,E2 -14344.017} C_VEL
LIN {X 0,Y 343.939,Z 590.002,A -85,B 0,C 180,E1 -14345.18,E2 -14345.18} C_VEL
LIN {X 0,Y 340.898,Z 582.713,A -85,B 0,C 180,E1 -14345.972,E2 -14345.972} C_VEL
LIN {X 0,Y 342.227,Z 590.419,A -85,B 0,C 180,E1 -14349.538,E2 -14349.538} C_VEL
LIN {X 0,Y 342.559,Z 595.186,A -85,B 0,C 180,E1 -14351.7,E2 -14351.7} C_VEL
LIN {X 0,Y 342.267,Z 602.651,A -85,B 0,C 180,E1 -14354.994,E2 -14354.994} C_VEL
LIN {X 0,Y 341.84,Z 610.176,A -85,B 0,C 180,E1 -14358.281,E2 -14358.281} C_VEL
LIN {X 0,Y 341.646,Z 616.061,A -85,B 0,C 180,E1 -14360.869,E2 -14360.869} C_VEL
LIN {X 0,Y 340.925,Z 618.267,A -85,B 0,C 180,E1 -14361.781,E2 -14361.781} C_VEL
LIN {X 0,Y 337.973,Z 622.061,A -85,B 0,C 180,E1 -14363.244,E2 -14363.244} C_VEL
LIN {X 0,Y 335.449,Z 625.149,A -85,B 0,C 180,E1 -14364.424,E2 -14364.424} C_VEL
